LIN {X 0,Y 298.495,Z 251.301,A -85,B 0,C 180,E1 -16396.412,E2 -16396.412} C_VEL
LIN {X 0,Y 298.486,Z 251.3,A -85,B 0,C 180,E1 -16399.636,E2 -16399.636} C_VEL
LIN {X 0,Y 298.389,Z 251.313,A -85,B 0,C 180,E1 -16403.604,E2 -16403.604} C_VEL
LIN {X 0,Y 298.41,Z 251.315,A -85,B 0,C 180,E1 -16406.582,E2 -16406.582} C_VEL
LIN {X 0,Y 298.369,Z 251.315,A -85,B 0,C 180,E1 -16409.647,E2 -16409.647} C_VEL
LIN {X 0,Y 298.401,Z 251.314,A -85,B 0,C 180,E1 -16412.8,E2 -16412.8} C_VEL
LIN {X 0,Y 298.454,Z 251.307,A -85,B 0,C 180,E1 -16416.807,E2 -16416.807} C_VEL
LIN {X 0,Y 298.395,Z 251.314,A -85,B 0,C 180,E1 -16421.087,E2 -16421.087} C_VEL
LIN {X 0,Y 298.407,Z 251.311,A -85,B 0,C 180,E1 -16423.102,E2 -16423.102} C_VEL
LIN {X 0,Y 298.377,Z 251.316,A -85,B 0,C 180,E1 -16426.914,E2 -16426.914} C_VEL
LIN {X 0,Y 298.358,Z 251.318,A -85,B 0,C 180,E1 -16431.018,E2 -16431.018} C_VEL
LIN {X 0,Y 298.41,Z 251.316,A -85,B 0,C 180,E1 -16433.927,E2 -16433.927} C_VEL
LIN {X 0,Y 298.349,Z 251.319,A -85,B 0,C 180,E1 -16437.192,E2 -16437.192} C_VEL
LIN {X 0,Y 298.079,Z 251.351,A -85,B 0,C 180,E1 -16440.736,E2 -16440.736} C_VEL
LIN {X 0,Y 297.924,Z 251.374,A -85,B 0,C 180,E1 -16441.847,E2 -16441.847} C_VEL
LIN {X 0,Y 297.795,Z 253.558,A -85,B 0,C 180,E1 -16444.86,E2 -16444.86} C_VEL
LIN {X 0,Y 297.677,Z 255.967,A -85,B 0,C 180,E1 -16447.804,E2 -16447.804} C_VEL
LIN {X 0,Y 297.6,Z 258.252,A -85,B 0,C 180,E1 -16450.465,E2 -16450.465} C_VEL
LIN {X 0,Y 301.663,Z 271.623,A -85,B 0,C 180,E1 -16451.421,E2 -16451.421} C_VEL
LIN {X 0,Y 304.774,Z 284.38,A -85,B 0,C 180,E1 -16452.554,E2 -16452.554} C_VEL
LIN {X 0,Y 306.16,Z 292.534,A -85,B 0,C 180,E1 -16453.404,E2 -16453.404} C_VEL
LIN {X 0,Y 304.897,Z 304.106,A -85,B 0,C 180,E1 -16454.626,E2 -16454.626} C_VEL
LIN {X 0,Y 303.62,Z 314.955,A -85,B 0,C 180,E1 -16456.102,E2 -16456.102} C_VEL
LIN {X 0,Y 302.035,Z 325.56,A -85,B 0,C 180,E1 -16457.91,E2 -16457.91} C_VEL
LIN {X 0,Y 300.876,Z 333.375,A -85,B 0,C 180,E1 -16459.568,E2 -16459.568} C_VEL
LIN {X 0,Y 299.75,Z 341.018,A -85,B 0,C 180,E1 -16461.572,E2 -16461.572} C_VEL
LIN {X 0,Y 298.938,Z 346.239,A -85,B 0,C 180,E1 -16463.247,E2 -16463.247} C_VEL
LIN {X 0,Y 297.998,Z 351.328,A -85,B 0,C 180,E1 -16465.263,E2 -16465.263} C_VEL
LIN {X 0,Y 297.426,Z 355.273,A -85,B 0,C 180,E1 -16467.289,E2 -16467.289} C_VEL
LIN {X 0,Y 297.194,Z 357.306,A -85,B 0,C 180,E1 -16468.643,E2 -16468.643} C_VEL
LIN {X 0,Y 297.056,Z 358.924,A -85,B 0,C 180,E1 -16469.998,E2 -16469.998} C_VEL
LIN {X 0,Y 296.954,Z 360.15,A -85,B 0,C 180,E1 -16471.354,E2 -16471.354} C_VEL
LIN {X 0,Y 296.857,Z 360.979,A -85,B 0,C 180,E1 -16472.712,E2 -16472.712} C_VEL
LIN {X 0,Y 296.97,Z 361.408,A -85,B 0,C 180,E1 -16475.43,E2 -16475.43} C_VEL
LIN {X 0,Y 297.058,Z 361.061,A -85,B 0,C 180,E1 -16476.792,E2 -16476.792} C_VEL
LIN {X 0,Y 297.19,Z 360.323,A -85,B 0,C 180,E1 -16478.155,E2 -16478.155} C_VEL
LIN {X 0,Y 297.693,Z 357.573,A -85,B 0,C 180,E1 -16480.884,E2 -16480.884} C_VEL
LIN {X 0,Y 298.353,Z 354.392,A -85,B 0,C 180,E1 -16482.929,E2 -16482.929} C_VEL
LIN {X 0,Y 299.246,Z 350.14,A -85,B 0,C 180,E1 -16484.97,E2 -16484.97} C_VEL
LIN {X 0,Y 300.406,Z 344.691,A -85,B 0,C 180,E1 -16487.002,E2 -16487.002} C_VEL
LIN {X 0,Y 301.868,Z 337.861,A -85,B 0,C 180,E1 -16489.021,E2 -16489.021} C_VEL
LIN {X 0,Y 303.56,Z 329.278,A -85,B 0,C 180,E1 -16491.028,E2 -16491.028} C_VEL
LIN {X 0,Y 305.117,Z 320.347,A -85,B 0,C 180,E1 -16492.71,E2 -16492.71} C_VEL
LIN {X 0,Y 306.776,Z 310.709,A -85,B 0,C 180,E1 -16494.171,E2 -16494.171} C_VEL
LIN {X 0,Y 308.399,Z 299.995,A -85,B 0,C 180,E1 -16495.474,E2 -16495.474} C_VEL
LIN {X 0,Y 308.698,Z 295.769,A -85,B 0,C 180,E1 -16495.93,E2 -16495.93} C_VEL
LIN {X 0,Y 306.296,Z 284.543,A -85,B 0,C 180,E1 -16497.236,E2 -16497.236} C_VEL
LIN {X 0,Y 302.82,Z 272.388,A -85,B 0,C 180,E1 -16498.45,E2 -16498.45} C_VEL
LIN {X 0,Y 298.604,Z 261.16,A -85,B 0,C 180,E1 -16499.443,E2 -16499.443} C_VEL
LIN {X 0,Y 297.888,Z 258.687,A -85,B 0,C 180,E1 -16499.656,E2 -16499.656} C_VEL
LIN {X 0,Y 298.06,Z 256.149,A -85,B 0,C 180,E1 -16502.839,E2 -16502.839} C_VEL
LIN {X 0,Y 298.264,Z 253.165,A -85,B 0,C 180,E1 -16506.76,E2 -16506.76} C_VEL
LIN {X 0,Y 298.264,Z 251.331,A -85,B 0,C 180,E1 -16509.506,E2 -16509.506} C_VEL
LIN {X 0,Y 298.363,Z 251.321,A -85,B 0,C 180,E1 -16513.095,E2 -16513.095} C_VEL
LIN {X 0,Y 298.396,Z 251.317,A -85,B 0,C 180,E1 -16516.919,E2 -16516.919} C_VEL
LIN {X 0,Y 298.407,Z 251.314,A -85,B 0,C 180,E1 -16521.002,E2 -16521.002} C_VEL
LIN {X 0,Y 298.424,Z 251.31,A -85,B 0,C 180,E1 -16523.931,E2 -16523.931} C_VEL
LIN {X 0,Y 298.384,Z 251.317,A -85,B 0,C 180,E1 -16527.982,E2 -16527.982} C_VEL
LIN {X 0,Y 298.449,Z 251.307,A -85,B 0,C 180,E1 -16531.903,E2 -16531.903} C_VEL
LIN {X 0,Y 298.476,Z 251.305,A -85,B 0,C 180,E1 -16534.923,E2 -16534.923} C_VEL
LIN {X 0,Y 298.44,Z 251.31,A -85,B 0,C 180,E1 -16539.314,E2 -16539.314} C_VEL
LIN {X 0,Y 298.527,Z 251.299,A -85,B 0,C 180,E1 -16542.178,E2 -16542.178} C_VEL
LIN {X 0,Y 298.539,Z 251.294,A -85,B 0,C 180,E1 -16545.707,E2 -16545.707} C_VEL
LIN {X 0,Y 298.582,Z 251.294,A -85,B 0,C 180,E1 -16549.146,E2 -16549.146} C_VEL
LIN {X 0,Y 298.744,Z 251.272,A -85,B 0,C 180,E1 -16551.565,E2 -16551.565} C_VEL
LIN {X 0,Y 298.09,Z 251.356,A -85,B 0,C 180,E1 -16552.688,E2 -16552.688} C_VEL
LIN {X 0,Y 295.26,Z 251.712,A -85,B 0,C 180,E1 -16554.517,E2 -16554.517} C_VEL
LIN {X 0,Y 292.869,Z 252.008,A -85,B 0,C 180,E1 -16556.002,E2 -16556.002} C_VEL
LIN {X 0,Y 291.865,Z 252.131,A -85,B 0,C 180,E1 -16557.151,E2 -16557.151} C_VEL
LIN {X 0,Y 291.795,Z 252.137,A -85,B 0,C 180,E1 -16557.54,E2 -16557.54} C_VEL
LIN {X 0,Y 291.941,Z 252.12,A -85,B 0,C 180,E1 -16560,E2 -16560} C_VEL
LIN {X 0,Y 291.781,Z 252.14,A -85,B 0,C 180,E1 -16562.761,E2 -16562.761} C_VEL
LIN {X 0,Y 291.738,Z 252.145,A -85,B 0,C 180,E1 -16566.918,E2 -16566.918} C_VEL
LIN {X 0,Y 291.618,Z 252.16,A -85,B 0,C 180,E1 -16569.712,E2 -16569.712} C_VEL
LIN {X 0,Y 291.511,Z 252.173,A -85,B 0,C 180,E1 -16573.951,E2 -16573.951} C_VEL
LIN {X 0,Y 291.476,Z 252.176,A -85,B 0,C 180,E1 -16576.818,E2 -16576.818} C_VEL
LIN {X 0,Y 291.44,Z 252.179,A -85,B 0,C 180,E1 -16579.876,E2 -16579.876} C_VEL
LIN {X 0,Y 291.39,Z 252.188,A -85,B 0,C 180,E1 -16584.206,E2 -16584.206} C_VEL
LIN {X 0,Y 291.415,Z 252.185,A -85,B 0,C 180,E1 -16587.272,E2 -16587.272} C_VEL
LIN {X 0,Y 291.331,Z 252.197,A -85,B 0,C 180,E1 -16590.437,E2 -16590.437} C_VEL
LIN {X 0,Y 291.336,Z 252.196,A -85,B 0,C 180,E1 -16593.699,E2 -16593.699} C_VEL
LIN {X 0,Y 291.416,Z 252.319,A -85,B 0,C 180,E1 -16596.863,E2 -16596.863} C_VEL
LIN {X 0,Y 292.017,Z 256.126,A -85,B 0,C 180,E1 -16600.527,E2 -16600.527} C_VEL
LIN {X 0,Y 292.801,Z 260.152,A -85,B 0,C 180,E1 -16604.113,E2 -16604.113} C_VEL
LIN {X 0,Y 293.64,Z 264.805,A -85,B 0,C 180,E1 -16607.924,E2 -16607.924} C_VEL
LIN {X 0,Y 294.327,Z 268.492,A -85,B 0,C 180,E1 -16610.771,E2 -16610.771} C_VEL
LIN {X 0,Y 294.514,Z 272.114,A -85,B 0,C 180,E1 -16613.378,E2 -16613.378} C_VEL
LIN {X 0,Y 293.527,Z 277.438,A -85,B 0,C 180,E1 -16616.931,E2 -16616.931} C_VEL
LIN {X 0,Y 292.414,Z 284.163,A -85,B 0,C 180,E1 -16621.272,E2 -16621.272} C_VEL
LIN {X 0,Y 291.705,Z 288.494,A -85,B 0,C 180,E1 -16624.014,E2 -16624.014} C_VEL
LIN {X 0,Y 295.156,Z 303.237,A -85,B 0,C 180,E1 -16625.062,E2 -16625.062} C_VEL
LIN {X 0,Y 297.245,Z 315.455,A -85,B 0,C 180,E1 -16626.118,E2 -16626.118} C_VEL
LIN {X 0,Y 298.415,Z 327.56,A -85,B 0,C 180,E1 -16627.354,E2 -16627.354} C_VEL
LIN {X 0,Y 298.729,Z 339.369,A -85,B 0,C 180,E1 -16628.797,E2 -16628.797} C_VEL
LIN {X 0,Y 296.902,Z 350.121,A -85,B 0,C 180,E1 -16630.289,E2 -16630.289} C_VEL
LIN {X 0,Y 295.152,Z 359.818,A -85,B 0,C 180,E1 -16631.97,E2 -16631.97} C_VEL
LIN {X 0,Y 293.752,Z 367.79,A -85,B 0,C 180,E1 -16633.675,E2 -16633.675} C_VEL
LIN {X 0,Y 292.298,Z 375.615,A -85,B 0,C 180,E1 -16635.735,E2 -16635.735} C_VEL
LIN {X 0,Y 290.944,Z 382.812,A -85,B 0,C 180,E1 -16638.154,E2 -16638.154} C_VEL
LIN {X 0,Y 290.222,Z 387.639,A -85,B 0,C 180,E1 -16640.243,E2 -16640.243} C_VEL
LIN {X 0,Y 289.804,Z 391.357,A -85,B 0,C 180,E1 -16642.337,E2 -16642.337} C_VEL
LIN {X 0,Y 289.624,Z 394.066,A -85,B 0,C 180,E1 -16644.432,E2 -16644.432} C_VEL
LIN {X 0,Y 289.579,Z 395.353,A -85,B 0,C 180,E1 -16645.827,E2 -16645.827} C_VEL
LIN {X 0,Y 289.548,Z 396.233,A -85,B 0,C 180,E1 -16647.22,E2 -16647.22} C_VEL
LIN {X 0,Y 289.693,Z 396.729,A -85,B 0,C 180,E1 -16650.002,E2 -16650.002} C_VEL
LIN {X 0,Y 289.608,Z 396.378,A -85,B 0,C 180,E1 -16651.393,E2 -16651.393} C_VEL
LIN {X 0,Y 289.568,Z 395.633,A -85,B 0,C 180,E1 -16652.784,E2 -16652.784} C_VEL
LIN {X 0,Y 289.605,Z 394.441,A -85,B 0,C 180,E1 -16654.177,E2 -16654.177} C_VEL
LIN {X 0,Y 289.638,Z 392.512,A -85,B 0,C 180,E1 -16655.813,E2 -16655.813} C_VEL
LIN {X 0,Y 289.919,Z 388.286,A -85,B 0,C 180,E1 -16658.365,E2 -16658.365} C_VEL
LIN {X 0,Y 290.444,Z 383.58,A -85,B 0,C 180,E1 -16660.458,E2 -16660.458} C_VEL
LIN {X 0,Y 291.385,Z 376.481,A -85,B 0,C 180,E1 -16662.893,E2 -16662.893} C_VEL
LIN {X 0,Y 292.543,Z 368.803,A -85,B 0,C 180,E1 -16664.969,E2 -16664.969} C_VEL
LIN {X 0,Y 293.742,Z 360.95,A -85,B 0,C 180,E1 -16666.687,E2 -16666.687} C_VEL
LIN {X 0,Y 295.134,Z 351.353,A -85,B 0,C 180,E1 -16668.394,E2 -16668.394} C_VEL
LIN {X 0,Y 296.77,Z 340.732,A -85,B 0,C 180,E1 -16669.905,E2 -16669.905} C_VEL
LIN {X 0,Y 297.183,Z 336.584,A -85,B 0,C 180,E1 -16670.417,E2 -16670.417} C_VEL
LIN {X 0,Y 296.404,Z 324.766,A -85,B 0,C 180,E1 -16671.772,E2 -16671.772} C_VEL
LIN {X 0,Y 295.302,Z 312.997,A -85,B 0,C 180,E1 -16672.858,E2 -16672.858} C_VEL
LIN {X 0,Y 293.429,Z 300.224,A -85,B 0,C 180,E1 -16673.794,E2 -16673.794} C_VEL
LIN {X 0,Y 291.24,Z 288.858,A -85,B 0,C 180,E1 -16674.459,E2 -16674.459} C_VEL
LIN {X 0,Y 292.173,Z 281.913,A -85,B 0,C 180,E1 -16678.758,E2 -16678.758} C_VEL
LIN {X 0,Y 293.275,Z 275.145,A -85,B 0,C 180,E1 -16682.993,E2 -16682.993} C_VEL
LIN {X 0,Y 293.926,Z 271.096,A -85,B 0,C 180,E1 -16685.613,E2 -16685.613} C_VEL
LIN {X 0,Y 294.053,Z 267.61,A -85,B 0,C 180,E1 -16687.934,E2 -16687.934} C_VEL
LIN {X 0,Y 293.376,Z 263.132,A -85,B 0,C 180,E1 -16691.125,E2 -16691.125} C_VEL
LIN {X 0,Y 292.462,Z 258.16,A -85,B 0,C 180,E1 -16694.976,E2 -16694.976} C_VEL
LIN {X 0,Y 291.512,Z 252.834,A -85,B 0,C 180,E1 -16699.388,E2 -16699.388} C_VEL
LIN {X 0,Y 291.377,Z 252.193,A -85,B 0,C 180,E1 -16700.006,E2 -16700.006} C_VEL
LIN {X 0,Y 291.411,Z 252.187,A -85,B 0,C 180,E1 -16702.92,E2 -16702.92} C_VEL
LIN {X 0,Y 291.351,Z 252.194,A -85,B 0,C 180,E1 -16706.302,E2 -16706.302} C_VEL
LIN {X 0,Y 291.377,Z 252.191,A -85,B 0,C 180,E1 -16710.267,E2 -16710.267} C_VEL
LIN {X 0,Y 291.385,Z 252.19,A -85,B 0,C 180,E1 -16714.269,E2 -16714.269} C_VEL
LIN {X 0,Y 291.379,Z 252.187,A -85,B 0,C 180,E1 -16717.299,E2 -16717.299} C_VEL
LIN {X 0,Y 291.414,Z 252.187,A -85,B 0,C 180,E1 -16720.267,E2 -16720.267} C_VEL
LIN {X 0,Y 291.482,Z 252.176,A -85,B 0,C 180,E1 -16724.683,E2 -16724.683} C_VEL
LIN {X 0,Y 291.534,Z 252.169,A -85,B 0,C 180,E1 -16728.881,E2 -16728.881} C_VEL
LIN {X 0,Y 291.676,Z 252.155,A -85,B 0,C 180,E1 -16731.688,E2 -16731.688} C_VEL
LIN {X 0,Y 291.63,Z 252.157,A -85,B 0,C 180,E1 -16734.468,E2 -16734.468} C_VEL
LIN {X 0,Y 291.895,Z 252.123,A -85,B 0,C 180,E1 -16738.621,E2 -16738.621} C_VEL
LIN {X 0,Y 291.889,Z 252.126,A -85,B 0,C 180,E1 -16741.38,E2 -16741.38} C_VEL
LIN {X 0,Y 291.693,Z 252.15,A -85,B 0,C 180,E1 -16746.919,E2 -16746.919} C_VEL
LIN {X 0,Y 291.577,Z 252.162,A -85,B 0,C 180,E1 -16749.714,E2 -16749.714} C_VEL
LIN {X 0,Y 291.524,Z 252.168,A -85,B 0,C 180,E1 -16753.95,E2 -16753.95} C_VEL
LIN {X 0,Y 291.442,Z 252.182,A -85,B 0,C 180,E1 -16756.821,E2 -16756.821} C_VEL
LIN {X 0,Y 291.433,Z 252.178,A -85,B 0,C 180,E1 -16759.86,E2 -16759.86} C_VEL
LIN {X 0,Y 291.334,Z 252.193,A -85,B 0,C 180,E1 -16764.211,E2 -16764.211} C_VEL
LIN {X 0,Y 291.34,Z 252.193,A -85,B 0,C 180,E1 -16767.28,E2 -16767.28} C_VEL
LIN {X 0,Y 291.312,Z 252.198,A -85,B 0,C 180,E1 -16770.44,E2 -16770.44} C_VEL
LIN {X 0,Y 291.352,Z 252.19,A -85,B 0,C 180,E1 -16773.698,E2 -16773.698} C_VEL
LIN {X 0,Y 291.384,Z 252.186,A -85,B 0,C 180,E1 -16777.253,E2 -16777.253} C_VEL
LIN {X 0,Y 291.34,Z 252.195,A -85,B 0,C 180,E1 -16780.642,E2 -16780.642} C_VEL
LIN {X 0,Y 291.298,Z 252.2,A -85,B 0,C 180,E1 -16784.401,E2 -16784.401} C_VEL
LIN {X 0,Y 291.301,Z 252.2,A -85,B 0,C 180,E1 -16788.411,E2 -16788.411} C_VEL
LIN {X 0,Y 291.392,Z 252.186,A -85,B 0,C 180,E1 -16792.915,E2 -16792.915} C_VEL
LIN {X 0,Y 291.328,Z 252.194,A -85,B 0,C 180,E1 -16796.297,E2 -16796.297} C_VEL
LIN {X 0,Y 291.106,Z 252.221,A -85,B 0,C 180,E1 -16799.534,E2 -16799.534} C_VEL
LIN {X 0,Y 290.966,Z 252.238,A -85,B 0,C 180,E1 -16801.111,E2 -16801.111} C_VEL
LIN {X 0,Y 290.841,Z 252.791,A -85,B 0,C 180,E1 -16802.667,E2 -16802.667} C_VEL
LIN {X 0,Y 290.667,Z 256.033,A -85,B 0,C 180,E1 -16806.752,E2 -16806.752} C_VEL
LIN {X 0,Y 290.568,Z 258.744,A -85,B 0,C 180,E1 -16809.906,E2 -16809.906} C_VEL
LIN {X 0,Y 294.61,Z 271.745,A -85,B 0,C 180,E1 -16810.872,E2 -16810.872} C_VEL
LIN {X 0,Y 297.663,Z 283.982,A -85,B 0,C 180,E1 -16811.988,E2 -16811.988} C_VEL
LIN {X 0,Y 299.429,Z 293.541,A -85,B 0,C 180,E1 -16813.017,E2 -16813.017} C_VEL
LIN {X 0,Y 298.114,Z 305.01,A -85,B 0,C 180,E1 -16814.268,E2 -16814.268} C_VEL
LIN {X 0,Y 296.773,Z 315.748,A -85,B 0,C 180,E1 -16815.775,E2 -16815.775} C_VEL
LIN {X 0,Y 295.139,Z 326.292,A -85,B 0,C 180,E1 -16817.623,E2 -16817.623} C_VEL
LIN {X 0,Y 293.944,Z 334.054,A -85,B 0,C 180,E1 -16819.32,E2 -16819.32} C_VEL
LIN {X 0,Y 292.75,Z 341.637,A -85,B 0,C 180,E1 -16821.369,E2 -16821.369} C_VEL
LIN {X 0,Y 291.525,Z 348.63,A -85,B 0,C 180,E1 -16823.77,E2 -16823.77} C_VEL
LIN {X 0,Y 290.747,Z 353.286,A -85,B 0,C 180,E1 -16825.839,E2 -16825.839} C_VEL
LIN {X 0,Y 290.225,Z 356.849,A -85,B 0,C 180,E1 -16827.916,E2 -16827.916} C_VEL
LIN {X 0,Y 289.981,Z 359.412,A -85,B 0,C 180,E1 -16829.998,E2 -16829.998} C_VEL
LIN {X 0,Y 289.861,Z 360.626,A -85,B 0,C 180,E1 -16831.387,E2 -16831.387} C_VEL
LIN {X 0,Y 289.772,Z 361.427,A -85,B 0,C 180,E1 -16832.778,E2 -16832.778} C_VEL
LIN {X 0,Y 289.906,Z 361.828,A -85,B 0,C 180,E1 -16835.563,E2 -16835.563} C_VEL
LIN {X 0,Y 289.996,Z 361.469,A -85,B 0,C 180,E1 -16836.958,E2 -16836.958} C_VEL
LIN {X 0,Y 290.128,Z 360.706,A -85,B 0,C 180,E1 -16838.355,E2 -16838.355} C_VEL
LIN {X 0,Y 290.68,Z 357.926,A -85,B 0,C 180,E1 -16841.15,E2 -16841.15} C_VEL
LIN {X 0,Y 291.399,Z 354.714,A -85,B 0,C 180,E1 -16843.243,E2 -16843.243} C_VEL
LIN {X 0,Y 292.34,Z 350.43,A -85,B 0,C 180,E1 -16845.332,E2 -16845.332} C_VEL
LIN {X 0,Y 293.568,Z 344.946,A -85,B 0,C 180,E1 -16847.41,E2 -16847.41} C_VEL
LIN {X 0,Y 295.116,Z 338.074,A -85,B 0,C 180,E1 -16849.473,E2 -16849.473} C_VEL
LIN {X 0,Y 296.91,Z 329.424,A -85,B 0,C 180,E1 -16851.522,E2 -16851.522} C_VEL
LIN {X 0,Y 298.437,Z 321.024,A -85,B 0,C 180,E1 -16853.137,E2 -16853.137} C_VEL
LIN {X 0,Y 300.28,Z 310.729,A -85,B 0,C 180,E1 -16854.729,E2 -16854.729} C_VEL
LIN {X 0,Y 301.951,Z 299.88,A -85,B 0,C 180,E1 -16856.058,E2 -16856.058} C_VEL
LIN {X 0,Y 302.019,Z 296.95,A -85,B 0,C 180,E1 -16856.394,E2 -16856.394} C_VEL
LIN {X 0,Y 299.713,Z 286.068,A -85,B 0,C 180,E1 -16857.723,E2 -16857.723} C_VEL
LIN {X 0,Y 296.345,Z 274.182,A -85,B 0,C 180,E1 -16858.977,E2 -16858.977} C_VEL
LIN {X 0,Y 291.861,Z 262.102,A -85,B 0,C 180,E1 -16860.099,E2 -16860.099} C_VEL
LIN {X 0,Y 290.879,Z 259.15,A -85,B 0,C 180,E1 -16860.354,E2 -16860.354} C_VEL
LIN {X 0,Y 291.079,Z 256.531,A -85,B 0,C 180,E1 -16863.731,E2 -16863.731} C_VEL
LIN {X 0,Y 291.249,Z 253.962,A -85,B 0,C 180,E1 -16867.22,E2 -16867.22} C_VEL
LIN {X 0,Y 291.257,Z 252.385,A -85,B 0,C 180,E1 -16869.452,E2 -16869.452} C_VEL
LIN {X 0,Y 291.277,Z 252.203,A -85,B 0,C 180,E1 -16872.497,E2 -16872.497} C_VEL
LIN {X 0,Y 291.302,Z 252.201,A -85,B 0,C 180,E1 -16876.364,E2 -16876.364} C_VEL
LIN {X 0,Y 291.379,Z 252.191,A -85,B 0,C 180,E1 -16880.515,E2 -16880.515} C_VEL
LIN {X 0,Y 291.417,Z 252.183,A -85,B 0,C 180,E1 -16882.921,E2 -16882.921} C_VEL
LIN {X 0,Y 291.336,Z 252.192,A -85,B 0,C 180,E1 -16886.3,E2 -16886.3} C_VEL
LIN {X 0,Y 291.374,Z 252.189,A -85,B 0,C 180,E1 -16890.26,E2 -16890.26} C_VEL
LIN {X 0,Y 291.405,Z 252.189,A -85,B 0,C 180,E1 -16894.271,E2 -16894.271} C_VEL
LIN {X 0,Y 291.372,Z 252.191,A -85,B 0,C 180,E1 -16897.298,E2 -16897.298} C_VEL
LIN {X 0,Y 291.448,Z 252.181,A -85,B 0,C 180,E1 -16900.269,E2 -16900.269} C_VEL
LIN {X 0,Y 291.545,Z 252.169,A -85,B 0,C 180,E1 -16904.623,E2 -16904.623} C_VEL
LIN {X 0,Y 291.526,Z 252.171,A -85,B 0,C 180,E1 -16908.88,E2 -16908.88} C_VEL
LIN {X 0,Y 291.7,Z 252.15,A -85,B 0,C 180,E1 -16911.688,E2 -16911.688} C_VEL
LIN {X 0,Y 291.625,Z 252.16,A -85,B 0,C 180,E1 -16914.468,E2 -16914.468} C_VEL
LIN {X 0,Y 291.795,Z 252.137,A -85,B 0,C 180,E1 -16917.54,E2 -16917.54} C_VEL
LIN {X 0,Y 291.168,Z 252.217,A -85,B 0,C 180,E1 -16918.694,E2 -16918.694} C_VEL
LIN {X 0,Y 288.341,Z 252.569,A -85,B 0,C 180,E1 -16920.573,E2 -16920.573} C_VEL
LIN {X 0,Y 284.987,Z 252.986,A -85,B 0,C 180,E1 -16922.88,E2 -16922.88} C_VEL
LIN {X 0,Y 284.575,Z 253.034,A -85,B 0,C 180,E1 -16923.679,E2 -16923.679} C_VEL
LIN {X 0,Y 284.69,Z 253.023,A -85,B 0,C 180,E1 -16927.09,E2 -16927.09} C_VEL
LIN {X 0,Y 284.555,Z 253.04,A -85,B 0,C 180,E1 -16929.956,E2 -16929.956} C_VEL
LIN {X 0,Y 284.47,Z 253.048,A -85,B 0,C 180,E1 -16934.303,E2 -16934.303} C_VEL
LIN {X 0,Y 284.415,Z 253.058,A -85,B 0,C 180,E1 -16937.249,E2 -16937.249} C_VEL
LIN {X 0,Y 284.368,Z 253.063,A -85,B 0,C 180,E1 -16940.243,E2 -16940.243} C_VEL
LIN {X 0,Y 284.359,Z 253.065,A -85,B 0,C 180,E1 -16943.876,E2 -16943.876} C_VEL
LIN {X 0,Y 284.388,Z 253.06,A -85,B 0,C 180,E1 -16947.175,E2 -16947.175} C_VEL
LIN {X 0,Y 284.289,Z 253.073,A -85,B 0,C 180,E1 -16951.275,E2 -16951.275} C_VEL
LIN {X 0,Y 284.332,Z 253.064,A -85,B 0,C 180,E1 -16955.349,E2 -16955.349} C_VEL
LIN {X 0,Y 284.35,Z 253.206,A -85,B 0,C 180,E1 -16956.09,E2 -16956.09} C_VEL
LIN {X 0,Y 285.031,Z 257.246,A -85,B 0,C 180,E1 -16960.153,E2 -16960.153} C_VEL
LIN {X 0,Y 285.946,Z 262.067,A -85,B 0,C 180,E1 -16964.543,E2 -16964.543} C_VEL
LIN {X 0,Y 286.818,Z 266.953,A -85,B 0,C 180,E1 -16968.582,E2 -16968.582} C_VEL
LIN {X 0,Y 287.436,Z 270.659,A -85,B 0,C 180,E1 -16971.483,E2 -16971.483} C_VEL
LIN {X 0,Y 287.374,Z 273.855,A -85,B 0,C 180,E1 -16973.808,E2 -16973.808} C_VEL
LIN {X 0,Y 286.624,Z 277.769,A -85,B 0,C 180,E1 -16976.479,E2 -16976.479} C_VEL
LIN {X 0,Y 285.488,Z 283.813,A -85,B 0,C 180,E1 -16980.508,E2 -16980.508} C_VEL
LIN {X 0,Y 284.815,Z 288.181,A -85,B 0,C 180,E1 -16983.309,E2 -16983.309} C_VEL
LIN {X 0,Y 287.416,Z 298.87,A -85,B 0,C 180,E1 -16984.06,E2 -16984.06} C_VEL
LIN {X 0,Y 289.847,Z 311.024,A -85,B 0,C 180,E1 -16985.093,E2 -16985.093} C_VEL
LIN {X 0,Y 291.332,Z 322.541,A -85,B 0,C 180,E1 -16986.24,E2 -16986.24} C_VEL
LIN {X 0,Y 291.907,Z 333.646,A -85,B 0,C 180,E1 -16987.532,E2 -16987.532} C_VEL
LIN {X 0,Y 291.912,Z 340.559,A -85,B 0,C 180,E1 -16988.462,E2 -16988.462} C_VEL
LIN {X 0,Y 290.006,Z 351.033,A -85,B 0,C 180,E1 -16989.985,E2 -16989.985} C_VEL
LIN {X 0,Y 288.165,Z 360.713,A -85,B 0,C 180,E1 -16991.751,E2 -16991.751} C_VEL
LIN {X 0,Y 286.626,Z 368.947,A -85,B 0,C 180,E1 -16993.624,E2 -16993.624} C_VEL
LIN {X 0,Y 285.155,Z 376.45,A -85,B 0,C 180,E1 -16995.734,E2 -16995.734} C_VEL
LIN {X 0,Y 283.944,Z 382.493,A -85,B 0,C 180,E1 -16997.857,E2 -16997.857} C_VEL
LIN {X 0,Y 283.195,Z 387.297,A -85,B 0,C 180,E1 -16999.998,E2 -16999.998} C_VEL
LIN {X 0,Y 282.737,Z 390.993,A -85,B 0,C 180,E1 -17002.144,E2 -17002.144} C_VEL
LIN {X 0,Y 282.541,Z 393.682,A -85,B 0,C 180,E1 -17004.292,E2 -17004.292} C_VEL
LIN {X 0,Y 282.5,Z 394.959,A -85,B 0,C 180,E1 -17005.722,E2 -17005.722} C_VEL
LIN {X 0,Y 282.475,Z 395.824,A -85,B 0,C 180,E1 -17007.15,E2 -17007.15} C_VEL
LIN {X 0,Y 282.604,Z 396.297,A -85,B 0,C 180,E1 -17010.002,E2 -17010.002} C_VEL
LIN {X 0,Y 282.521,Z 395.936,A -85,B 0,C 180,E1 -17011.428,E2 -17011.428} C_VEL
LIN {X 0,Y 282.494,Z 395.177,A -85,B 0,C 180,E1 -17012.854,E2 -17012.854} C_VEL
LIN {X 0,Y 282.522,Z 393.968,A -85,B 0,C 180,E1 -17014.282,E2 -17014.282} C_VEL
LIN {X 0,Y 282.559,Z 392.251,A -85,B 0,C 180,E1 -17015.784,E2 -17015.784} C_VEL
LIN {X 0,Y 282.747,Z 389.076,A -85,B 0,C 180,E1 -17017.859,E2 -17017.859} C_VEL
LIN {X 0,Y 283.217,Z 384.731,A -85,B 0,C 180,E1 -17020.005,E2 -17020.005} C_VEL
LIN {X 0,Y 284.069,Z 378.16,A -85,B 0,C 180,E1 -17022.504,E2 -17022.504} C_VEL
LIN {X 0,Y 285.26,Z 370.955,A -85,B 0,C 180,E1 -17024.629,E2 -17024.629} C_VEL
LIN {X 0,Y 286.66,Z 361.977,A -85,B 0,C 180,E1 -17026.745,E2 -17026.745} C_VEL
LIN {X 0,Y 288.056,Z 352.767,A -85,B 0,C 180,E1 -17028.494,E2 -17028.494} C_VEL
LIN {X 0,Y 289.65,Z 342.578,A -85,B 0,C 180,E1 -17030.045,E2 -17030.045} C_VEL
LIN {X 0,Y 290.295,Z 337.231,A -85,B 0,C 180,E1 -17030.738,E2 -17030.738} C_VEL
LIN {X 0,Y 289.54,Z 325.291,A -85,B 0,C 180,E1 -17032.166,E2 -17032.166} C_VEL
LIN {X 0,Y 288.485,Z 313.149,A -85,B 0,C 180,E1 -17033.334,E2 -17033.334} C_VEL
LIN {X 0,Y 286.603,Z 300.298,A -85,B 0,C 180,E1 -17034.319,E2 -17034.319} C_VEL
LIN {X 0,Y 284.248,Z 288.415,A -85,B 0,C 180,E1 -17035.052,E2 -17035.052} C_VEL
LIN {X 0,Y 285.294,Z 281.424,A -85,B 0,C 180,E1 -17039.519,E2 -17039.519} C_VEL
LIN {X 0,Y 286.334,Z 275.364,A -85,B 0,C 180,E1 -17043.434,E2 -17043.434} C_VEL
LIN {X 0,Y 287.068,Z 270.268,A -85,B 0,C 180,E1 -17046.858,E2 -17046.858} C_VEL
LIN {X 0,Y 287.02,Z 268.038,A -85,B 0,C 180,E1 -17048.413,E2 -17048.413} C_VEL
LIN {X 0,Y 286.291,Z 263.878,A -85,B 0,C 180,E1 -17051.517,E2 -17051.517} C_VEL
LIN {X 0,Y 285.323,Z 258.682,A -85,B 0,C 180,E1 -17055.59,E2 -17055.59} C_VEL
LIN {X 0,Y 284.426,Z 253.592,A -85,B 0,C 180,E1 -17060.026,E2 -17060.026} C_VEL
LIN {X 0,Y 284.329,Z 253.07,A -85,B 0,C 180,E1 -17060.699,E2 -17060.699} C_VEL
LIN {X 0,Y 284.348,Z 253.067,A -85,B 0,C 180,E1 -17064.653,E2 -17064.653} C_VEL
LIN {X 0,Y 284.294,Z 253.072,A -85,B 0,C 180,E1 -17068.725,E2 -17068.725} C_VEL
LIN {X 0,Y 284.299,Z 253.071,A -85,B 0,C 180,E1 -17071.986,E2 -17071.986} C_VEL
LIN {X 0,Y 284.334,Z 253.069,A -85,B 0,C 180,E1 -17076.145,E2 -17076.145} C_VEL
LIN {X 0,Y 284.384,Z 253.062,A -85,B 0,C 180,E1 -17079.905,E2 -17079.905} C_VEL
LIN {X 0,Y 284.44,Z 253.054,A -85,B 0,C 180,E1 -17084.504,E2 -17084.504} C_VEL
LIN {X 0,Y 284.466,Z 253.05,A -85,B 0,C 180,E1 -17088.601,E2 -17088.601} C_VEL
LIN {X 0,Y 284.63,Z 253.031,A -85,B 0,C 180,E1 -17091.48,E2 -17091.48} C_VEL
LIN {X 0,Y 284.6,Z 253.033,A -85,B 0,C 180,E1 -17094.331,E2 -17094.331} C_VEL
LIN {X 0,Y 284.862,Z 252.999,A -85,B 0,C 180,E1 -17098.586,E2 -17098.586} C_VEL
LIN {X 0,Y 284.855,Z 253.002,A -85,B 0,C 180,E1 -17101.414,E2 -17101.414} C_VEL
LIN {X 0,Y 284.648,Z 253.028,A -85,B 0,C 180,E1 -17107.091,E2 -17107.091} C_VEL
LIN {X 0,Y 284.523,Z 253.04,A -85,B 0,C 180,E1 -17109.957,E2 -17109.957} C_VEL
LIN {X 0,Y 284.472,Z 253.046,A -85,B 0,C 180,E1 -17114.304,E2 -17114.304} C_VEL
LIN {X 0,Y 284.371,Z 253.063,A -85,B 0,C 180,E1 -17118.741,E2 -17118.741} C_VEL
LIN {X 0,Y 284.311,Z 253.068,A -85,B 0,C 180,E1 -17121.765,E2 -17121.765} C_VEL
LIN {X 0,Y 284.291,Z 253.072,A -85,B 0,C 180,E1 -17124.851,E2 -17124.851} C_VEL
LIN {X 0,Y 284.272,Z 253.073,A -85,B 0,C 180,E1 -17128.017,E2 -17128.017} C_VEL
LIN {X 0,Y 284.287,Z 253.071,A -85,B 0,C 180,E1 -17131.276,E2 -17131.276} C_VEL
LIN {X 0,Y 284.349,Z 253.063,A -85,B 0,C 180,E1 -17135.347,E2 -17135.347} C_VEL
LIN {X 0,Y 284.32,Z 253.069,A -85,B 0,C 180,E1 -17138.168,E2 -17138.168} C_VEL
LIN {X 0,Y 284.277,Z 253.076,A -85,B 0,C 180,E1 -17142.123,E2 -17142.123} C_VEL
LIN {X 0,Y 284.245,Z 253.08,A -85,B 0,C 180,E1 -17146.185,E2 -17146.185} C_VEL
LIN {X 0,Y 284.262,Z 253.078,A -85,B 0,C 180,E1 -17150.035,E2 -17150.035} C_VEL
LIN {X 0,Y 284.322,Z 253.069,A -85,B 0,C 180,E1 -17153.61,E2 -17153.61} C_VEL
LIN {X 0,Y 284.243,Z 253.076,A -85,B 0,C 180,E1 -17157.211,E2 -17157.211} C_VEL
LIN {X 0,Y 284.016,Z 253.103,A -85,B 0,C 180,E1 -17160.335,E2 -17160.335} C_VEL
LIN {X 0,Y 283.827,Z 253.24,A -85,B 0,C 180,E1 -17161.933,E2 -17161.933} C_VEL
LIN {X 0,Y 283.689,Z 255.673,A -85,B 0,C 180,E1 -17165.091,E2 -17165.091} C_VEL
LIN {X 0,Y 283.539,Z 258.972,A -85,B 0,C 180,E1 -17169.181,E2 -17169.181} C_VEL
LIN {X 0,Y 283.556,Z 259.174,A -85,B 0,C 180,E1 -17169.316,E2 -17169.316} C_VEL
LIN {X 0,Y 287.672,Z 272.213,A -85,B 0,C 180,E1 -17170.326,E2 -17170.326} C_VEL
LIN {X 0,Y 290.573,Z 283.578,A -85,B 0,C 180,E1 -17171.395,E2 -17171.395} C_VEL
LIN {X 0,Y 292.681,Z 294.583,A -85,B 0,C 180,E1 -17172.614,E2 -17172.614} C_VEL
LIN {X 0,Y 291.343,Z 305.891,A -85,B 0,C 180,E1 -17173.892,E2 -17173.892} C_VEL
LIN {X 0,Y 289.955,Z 316.54,A -85,B 0,C 180,E1 -17175.433,E2 -17175.433} C_VEL
LIN {X 0,Y 288.258,Z 327.021,A -85,B 0,C 180,E1 -17177.323,E2 -17177.323} C_VEL
LIN {X 0,Y 287.019,Z 334.726,A -85,B 0,C 180,E1 -17179.059,E2 -17179.059} C_VEL
LIN {X 0,Y 285.754,Z 342.255,A -85,B 0,C 180,E1 -17181.156,E2 -17181.156} C_VEL
LIN {X 0,Y 284.902,Z 347.416,A -85,B 0,C 180,E1 -17182.913,E2 -17182.913} C_VEL
LIN {X 0,Y 283.931,Z 352.426,A -85,B 0,C 180,E1 -17185.028,E2 -17185.028} C_VEL
LIN {X 0,Y 283.332,Z 356.311,A -85,B 0,C 180,E1 -17187.154,E2 -17187.154} C_VEL
LIN {X 0,Y 283.085,Z 358.309,A -85,B 0,C 180,E1 -17188.575,E2 -17188.575} C_VEL
LIN {X 0,Y 282.907,Z 359.901,A -85,B 0,C 180,E1 -17189.998,E2 -17189.998} C_VEL
LIN {X 0,Y 282.769,Z 361.101,A -85,B 0,C 180,E1 -17191.422,E2 -17191.422} C_VEL
LIN {X 0,Y 282.757,Z 362.248,A -85,B 0,C 180,E1 -17194.274,E2 -17194.274} C_VEL
LIN {X 0,Y 282.888,Z 362.109,A -85,B 0,C 180,E1 -17196.406,E2 -17196.406} C_VEL
LIN {X 0,Y 283.085,Z 361.085,A -85,B 0,C 180,E1 -17198.564,E2 -17198.564} C_VEL
LIN {X 0,Y 283.689,Z 358.277,A -85,B 0,C 180,E1 -17201.429,E2 -17201.429} C_VEL
LIN {X 0,Y 284.458,Z 355.036,A -85,B 0,C 180,E1 -17203.572,E2 -17203.572} C_VEL
LIN {X 0,Y 285.45,Z 350.72,A -85,B 0,C 180,E1 -17205.711,E2 -17205.711} C_VEL
LIN {X 0,Y 286.779,Z 345.2,A -85,B 0,C 180,E1 -17207.836,E2 -17207.836} C_VEL
LIN {X 0,Y 288.404,Z 338.28,A -85,B 0,C 180,E1 -17209.945,E2 -17209.945} C_VEL
LIN {X 0,Y 290.285,Z 329.571,A -85,B 0,C 180,E1 -17212.038,E2 -17212.038} C_VEL
LIN {X 0,Y 292.069,Z 320.038,A -85,B 0,C 180,E1 -17213.88,E2 -17213.88} C_VEL
LIN {X 0,Y 294.034,Z 309.492,A -85,B 0,C 180,E1 -17215.48,E2 -17215.48} C_VEL
LIN {X 0,Y 295.531,Z 299.762,A -85,B 0,C 180,E1 -17216.668,E2 -17216.668} C_VEL
LIN {X 0,Y 293.744,Z 289.959,A -85,B 0,C 180,E1 -17217.935,E2 -17217.935} C_VEL
LIN {X 0,Y 290.847,Z 278.963,A -85,B 0,C 180,E1 -17219.199,E2 -17219.199} C_VEL
LIN {X 0,Y 286.926,Z 267.736,A -85,B 0,C 180,E1 -17220.355,E2 -17220.355} C_VEL
LIN {X 0,Y 283.969,Z 259.916,A -85,B 0,C 180,E1 -17221.058,E2 -17221.058} C_VEL
LIN {X 0,Y 283.907,Z 259.616,A -85,B 0,C 180,E1 -17221.083,E2 -17221.083} C_VEL
LIN {X 0,Y 284.102,Z 256.907,A -85,B 0,C 180,E1 -17224.675,E2 -17224.675} C_VEL
LIN {X 0,Y 284.233,Z 254.407,A -85,B 0,C 180,E1 -17228.179,E2 -17228.179} C_VEL
LIN {X 0,Y 284.215,Z 253.157,A -85,B 0,C 180,E1 -17230.007,E2 -17230.007} C_VEL
LIN {X 0,Y 284.226,Z 253.082,A -85,B 0,C 180,E1 -17234.186,E2 -17234.186} C_VEL
LIN {X 0,Y 284.265,Z 253.078,A -85,B 0,C 180,E1 -17238.123,E2 -17238.123} C_VEL
LIN {X 0,Y 284.327,Z 253.069,A -85,B 0,C 180,E1 -17242.273,E2 -17242.273} C_VEL
LIN {X 0,Y 284.315,Z 253.07,A -85,B 0,C 180,E1 -17245.351,E2 -17245.351} C_VEL
LIN {X 0,Y 284.285,Z 253.071,A -85,B 0,C 180,E1 -17248.724,E2 -17248.724} C_VEL
LIN {X 0,Y 284.386,Z 253.056,A -85,B 0,C 180,E1 -17252.826,E2 -17252.826} C_VEL
LIN {X 0,Y 284.357,Z 253.064,A -85,B 0,C 180,E1 -17256.706,E2 -17256.706} C_VEL
LIN {X 0,Y 284.393,Z 253.059,A -85,B 0,C 180,E1 -17261.261,E2 -17261.261} C_VEL
LIN {X 0,Y 284.482,Z 253.049,A -85,B 0,C 180,E1 -17264.458,E2 -17264.458} C_VEL
LIN {X 0,Y 284.477,Z 253.049,A -85,B 0,C 180,E1 -17268.601,E2 -17268.601} C_VEL
LIN {X 0,Y 284.65,Z 253.027,A -85,B 0,C 180,E1 -17271.481,E2 -17271.481} C_VEL
LIN {X 0,Y 284.595,Z 253.036,A -85,B 0,C 180,E1 -17274.331,E2 -17274.331} C_VEL
LIN {X 0,Y 284.846,Z 253.004,A -85,B 0,C 180,E1 -17278.586,E2 -17278.586} C_VEL
LIN {X 0,Y 284.844,Z 253.005,A -85,B 0,C 180,E1 -17281.414,E2 -17281.414} C_VEL
LIN {X 0,Y 284.575,Z 253.034,A -85,B 0,C 180,E1 -17283.679,E2 -17283.679} C_VEL
LIN {X 0,Y 283.814,Z 253.131,A -85,B 0,C 180,E1 -17284.86,E2 -17284.86} C_VEL
LIN {X 0,Y 281.013,Z 253.48,A -85,B 0,C 180,E1 -17286.788,E2 -17286.788} C_VEL
LIN {X 0,Y 277.871,Z 253.872,A -85,B 0,C 180,E1 -17289.156,E2 -17289.156} C_VEL
LIN {X 0,Y 277.516,Z 253.916,A -85,B 0,C 180,E1 -17289.973,E2 -17289.973} C_VEL
LIN {X 0,Y 277.423,Z 253.925,A -85,B 0,C 180,E1 -17294.675,E2 -17294.675} C_VEL
LIN {X 0,Y 277.334,Z 253.933,A -85,B 0,C 180,E1 -17299.234,E2 -17299.234} C_VEL
LIN {X 0,Y 277.309,Z 253.942,A -85,B 0,C 180,E1 -17304.171,E2 -17304.171} C_VEL
LIN {X 0,Y 277.318,Z 253.942,A -85,B 0,C 180,E1 -17307.507,E2 -17307.507} C_VEL
LIN {X 0,Y 277.262,Z 253.95,A -85,B 0,C 180,E1 -17310.483,E2 -17310.483} C_VEL
LIN {X 0,Y 277.29,Z 254.004,A -85,B 0,C 180,E1 -17315.212,E2 -17315.212} C_VEL
LIN {X 0,Y 277.772,Z 256.966,A -85,B 0,C 180,E1 -17318.344,E2 -17318.344} C_VEL
LIN {X 0,Y 278.637,Z 261.717,A -85,B 0,C 180,E1 -17322.923,E2 -17322.923} C_VEL
LIN {X 0,Y 279.45,Z 266.114,A -85,B 0,C 180,E1 -17326.831,E2 -17326.831} C_VEL
LIN {X 0,Y 280.215,Z 270.228,A -85,B 0,C 180,E1 -17330.212,E2 -17330.212} C_VEL
LIN {X 0,Y 280.52,Z 273.902,A -85,B 0,C 180,E1 -17333.041,E2 -17333.041} C_VEL
LIN {X 0,Y 279.73,Z 278.075,A -85,B 0,C 180,E1 -17336.007,E2 -17336.007} C_VEL
LIN {X 0,Y 278.42,Z 284.649,A -85,B 0,C 180,E1 -17340.516,E2 -17340.516} C_VEL
LIN {X 0,Y 277.943,Z 287.616,A -85,B 0,C 180,E1 -17342.52,E2 -17342.52} C_VEL
LIN {X 0,Y 279.966,Z 295.863,A -85,B 0,C 180,E1 -17343.115,E2 -17343.115} C_VEL
LIN {X 0,Y 282.598,Z 307.959,A -85,B 0,C 180,E1 -17344.153,E2 -17344.153} C_VEL
LIN {X 0,Y 284.28,Z 319.461,A -85,B 0,C 180,E1 -17345.301,E2 -17345.301} C_VEL
LIN {X 0,Y 285.09,Z 330.223,A -85,B 0,C 180,E1 -17346.547,E2 -17346.547} C_VEL
LIN {X 0,Y 285.205,Z 340.459,A -85,B 0,C 180,E1 -17347.929,E2 -17347.929} C_VEL
LIN {X 0,Y 283.34,Z 350.877,A -85,B 0,C 180,E1 -17349.493,E2 -17349.493} C_VEL
LIN {X 0,Y 281.61,Z 359.409,A -85,B 0,C 180,E1 -17351.071,E2 -17351.071} C_VEL
LIN {X 0,Y 280.095,Z 367.304,A -85,B 0,C 180,E1 -17352.855,E2 -17352.855} C_VEL
LIN {X 0,Y 278.522,Z 375.036,A -85,B 0,C 180,E1 -17355.013,E2 -17355.013} C_VEL
LIN {X 0,Y 276.965,Z 382.177,A -85,B 0,C 180,E1 -17357.546,E2 -17357.546} C_VEL
LIN {X 0,Y 276.181,Z 386.957,A -85,B 0,C 180,E1 -17359.741,E2 -17359.741} C_VEL
LIN {X 0,Y 275.677,Z 390.63,A -85,B 0,C 180,E1 -17361.942,E2 -17361.942} C_VEL
LIN {X 0,Y 275.443,Z 393.481,A -85,B 0,C 180,E1 -17364.325,E2 -17364.325} C_VEL
LIN {X 0,Y 275.404,Z 395.414,A -85,B 0,C 180,E1 -17367.077,E2 -17367.077} C_VEL
LIN {X 0,Y 275.515,Z 395.865,A -85,B 0,C 180,E1 -17370.002,E2 -17370.002} C_VEL
LIN {X 0,Y 275.437,Z 395.494,A -85,B 0,C 180,E1 -17371.464,E2 -17371.464} C_VEL
LIN {X 0,Y 275.423,Z 394.719,A -85,B 0,C 180,E1 -17372.927,E2 -17372.927} C_VEL
LIN {X 0,Y 275.444,Z 393.496,A -85,B 0,C 180,E1 -17374.392,E2 -17374.392} C_VEL
LIN {X 0,Y 275.516,Z 390.886,A -85,B 0,C 180,E1 -17376.594,E2 -17376.594} C_VEL
LIN {X 0,Y 275.832,Z 387.251,A -85,B 0,C 180,E1 -17378.796,E2 -17378.796} C_VEL
LIN {X 0,Y 276.386,Z 382.492,A -85,B 0,C 180,E1 -17380.996,E2 -17380.996} C_VEL
LIN {X 0,Y 277.505,Z 375.343,A -85,B 0,C 180,E1 -17383.55,E2 -17383.55} C_VEL
LIN {X 0,Y 278.789,Z 367.59,A -85,B 0,C 180,E1 -17385.726,E2 -17385.726} C_VEL
LIN {X 0,Y 280.067,Z 359.646,A -85,B 0,C 180,E1 -17387.527,E2 -17387.527} C_VEL
LIN {X 0,Y 281.576,Z 349.949,A -85,B 0,C 180,E1 -17389.314,E2 -17389.314} C_VEL
LIN {X 0,Y 283.406,Z 339.221,A -85,B 0,C 180,E1 -17390.886,E2 -17390.886} C_VEL
LIN {X 0,Y 282.898,Z 328.305,A -85,B 0,C 180,E1 -17392.298,E2 -17392.298} C_VEL
LIN {X 0,Y 282.056,Z 316.913,A -85,B 0,C 180,E1 -17393.497,E2 -17393.497} C_VEL
LIN {X 0,Y 280.348,Z 303.846,A -85,B 0,C 180,E1 -17394.613,E2 -17394.613} C_VEL
LIN {X 0,Y 277.793,Z 290.55,A -85,B 0,C 180,E1 -17395.513,E2 -17395.513} C_VEL
LIN {X 0,Y 277.295,Z 288.027,A -85,B 0,C 180,E1 -17395.65,E2 -17395.65} C_VEL
LIN {X 0,Y 278.438,Z 280.937,A -85,B 0,C 180,E1 -17400.321,E2 -17400.321} C_VEL
LIN {X 0,Y 279.547,Z 274.649,A -85,B 0,C 180,E1 -17404.525,E2 -17404.525} C_VEL
LIN {X 0,Y 280.034,Z 271.038,A -85,B 0,C 180,E1 -17407.039,E2 -17407.039} C_VEL
LIN {X 0,Y 279.688,Z 267.247,A -85,B 0,C 180,E1 -17409.851,E2 -17409.851} C_VEL
LIN {X 0,Y 278.917,Z 263.133,A -85,B 0,C 180,E1 -17413.053,E2 -17413.053} C_VEL
LIN {X 0,Y 278.021,Z 258.271,A -85,B 0,C 180,E1 -17417.148,E2 -17417.148} C_VEL
LIN {X 0,Y 277.302,Z 253.945,A -85,B 0,C 180,E1 -17421.072,E2 -17421.072} C_VEL
LIN {X 0,Y 277.291,Z 253.946,A -85,B 0,C 180,E1 -17424.342,E2 -17424.342} C_VEL
LIN {X 0,Y 277.248,Z 253.949,A -85,B 0,C 180,E1 -17427.837,E2 -17427.837} C_VEL
LIN {X 0,Y 277.253,Z 253.947,A -85,B 0,C 180,E1 -17431.208,E2 -17431.208} C_VEL
LIN {X 0,Y 277.285,Z 253.946,A -85,B 0,C 180,E1 -17434.477,E2 -17434.477} C_VEL
LIN {X 0,Y 277.272,Z 253.946,A -85,B 0,C 180,E1 -17437.654,E2 -17437.654} C_VEL
LIN {X 0,Y 277.31,Z 253.941,A -85,B 0,C 180,E1 -17440.764,E2 -17440.764} C_VEL
LIN {X 0,Y 277.384,Z 253.932,A -85,B 0,C 180,E1 -17445.323,E2 -17445.323} C_VEL
LIN {X 0,Y 277.461,Z 253.926,A -85,B 0,C 180,E1 -17449.787,E2 -17449.787} C_VEL
LIN {X 0,Y 277.636,Z 253.898,A -85,B 0,C 180,E1 -17452.729,E2 -17452.729} C_VEL
LIN {X 0,Y 277.828,Z 253.876,A -85,B 0,C 180,E1 -17458.551,E2 -17458.551} C_VEL
LIN {X 0,Y 277.821,Z 253.878,A -85,B 0,C 180,E1 -17461.45,E2 -17461.45} C_VEL
LIN {X 0,Y 277.607,Z 253.907,A -85,B 0,C 180,E1 -17467.272,E2 -17467.272} C_VEL
LIN {X 0,Y 277.466,Z 253.918,A -85,B 0,C 180,E1 -17470.213,E2 -17470.213} C_VEL
LIN {X 0,Y 277.418,Z 253.926,A -85,B 0,C 180,E1 -17474.675,E2 -17474.675} C_VEL
LIN {X 0,Y 277.326,Z 253.938,A -85,B 0,C 180,E1 -17479.235,E2 -17479.235} C_VEL
LIN {X 0,Y 277.263,Z 253.944,A -85,B 0,C 180,E1 -17483.927,E2 -17483.927} C_VEL
LIN {X 0,Y 277.247,Z 253.948,A -85,B 0,C 180,E1 -17487.47,E2 -17487.47} C_VEL
LIN {X 0,Y 277.236,Z 253.951,A -85,B 0,C 180,E1 -17490.465,E2 -17490.465} C_VEL
LIN {X 0,Y 277.255,Z 253.946,A -85,B 0,C 180,E1 -17493.895,E2 -17493.895} C_VEL
LIN {X 0,Y 277.276,Z 253.944,A -85,B 0,C 180,E1 -17497.468,E2 -17497.468} C_VEL
LIN {X 0,Y 277.218,Z 253.952,A -85,B 0,C 180,E1 -17501.236,E2 -17501.236} C_VEL
LIN {X 0,Y 277.202,Z 253.953,A -85,B 0,C 180,E1 -17505.227,E2 -17505.227} C_VEL
LIN {X 0,Y 277.183,Z 253.957,A -85,B 0,C 180,E1 -17508.756,E2 -17508.756} C_VEL
LIN {X 0,Y 277.238,Z 253.951,A -85,B 0,C 180,E1 -17512.524,E2 -17512.524} C_VEL
LIN {X 0,Y 277.199,Z 253.955,A -85,B 0,C 180,E1 -17516.095,E2 -17516.095} C_VEL
LIN {X 0,Y 277.038,Z 253.973,A -85,B 0,C 180,E1 -17519.602,E2 -17519.602} C_VEL
LIN {X 0,Y 276.837,Z 253.997,A -85,B 0,C 180,E1 -17521.159,E2 -17521.159} C_VEL
LIN {X 0,Y 276.696,Z 256.144,A -85,B 0,C 180,E1 -17524.416,E2 -17524.416} C_VEL
LIN {X 0,Y 276.506,Z 259.524,A -85,B 0,C 180,E1 -17528.671,E2 -17528.671} C_VEL
LIN {X 0,Y 281.165,Z 274.053,A -85,B 0,C 180,E1 -17529.878,E2 -17529.878} C_VEL
LIN {X 0,Y 284.185,Z 286.351,A -85,B 0,C 180,E1 -17531.103,E2 -17531.103} C_VEL
LIN {X 0,Y 285.931,Z 295.627,A -85,B 0,C 180,E1 -17532.192,E2 -17532.192} C_VEL
LIN {X 0,Y 284.586,Z 306.754,A -85,B 0,C 180,E1 -17533.499,E2 -17533.499} C_VEL
LIN {X 0,Y 283.151,Z 317.326,A -85,B 0,C 180,E1 -17535.075,E2 -17535.075} C_VEL
LIN {X 0,Y 281.386,Z 327.738,A -85,B 0,C 180,E1 -17537.008,E2 -17537.008} C_VEL
LIN {X 0,Y 280.1,Z 335.388,A -85,B 0,C 180,E1 -17538.785,E2 -17538.785} C_VEL
LIN {X 0,Y 278.763,Z 342.872,A -85,B 0,C 180,E1 -17540.932,E2 -17540.932} C_VEL
LIN {X 0,Y 277.893,Z 347.996,A -85,B 0,C 180,E1 -17542.733,E2 -17542.733} C_VEL
LIN {X 0,Y 276.902,Z 352.973,A -85,B 0,C 180,E1 -17544.901,E2 -17544.901} C_VEL
LIN {X 0,Y 276.287,Z 356.827,A -85,B 0,C 180,E1 -17547.082,E2 -17547.082} C_VEL
LIN {X 0,Y 276.014,Z 358.811,A -85,B 0,C 180,E1 -17548.539,E2 -17548.539} C_VEL
LIN {X 0,Y 275.818,Z 360.39,A -85,B 0,C 180,E1 -17549.998,E2 -17549.998} C_VEL
LIN {X 0,Y 275.677,Z 361.573,A -85,B 0,C 180,E1 -17551.459,E2 -17551.459} C_VEL
LIN {X 0,Y 275.696,Z 362.681,A -85,B 0,C 180,E1 -17554.384,E2 -17554.384} C_VEL
LIN {X 0,Y 275.831,Z 362.558,A -85,B 0,C 180,E1 -17556.434,E2 -17556.434} C_VEL
LIN {X 0,Y 276.037,Z 361.466,A -85,B 0,C 180,E1 -17558.785,E2 -17558.785} C_VEL
LIN {X 0,Y 276.707,Z 358.629,A -85,B 0,C 180,E1 -17561.721,E2 -17561.721} C_VEL
LIN {X 0,Y 277.526,Z 355.358,A -85,B 0,C 180,E1 -17563.918,E2 -17563.918} C_VEL
LIN {X 0,Y 278.583,Z 351.011,A -85,B 0,C 180,E1 -17566.109,E2 -17566.109} C_VEL
LIN {X 0,Y 279.968,Z 345.457,A -85,B 0,C 180,E1 -17568.285,E2 -17568.285} C_VEL
LIN {X 0,Y 281.705,Z 338.481,A -85,B 0,C 180,E1 -17570.44,E2 -17570.44} C_VEL
LIN {X 0,Y 283.679,Z 329.72,A -85,B 0,C 180,E1 -17572.58,E2 -17572.58} C_VEL
LIN {X 0,Y 285.643,Z 319.793,A -85,B 0,C 180,E1 -17574.518,E2 -17574.518} C_VEL
LIN {X 0,Y 287.587,Z 309.476,A -85,B 0,C 180,E1 -17576.094,E2 -17576.094} C_VEL
LIN {X 0,Y 288.958,Z 301.226,A -85,B 0,C 180,E1 -17577.129,E2 -17577.129} C_VEL
LIN {X 0,Y 287.022,Z 290.726,A -85,B 0,C 180,E1 -17578.546,E2 -17578.546} C_VEL
LIN {X 0,Y 283.878,Z 278.999,A -85,B 0,C 180,E1 -17579.945,E2 -17579.945} C_VEL
LIN {X 0,Y 279.297,Z 266.254,A -85,B 0,C 180,E1 -17581.301,E2 -17581.301} C_VEL
LIN {X 0,Y 277.051,Z 260.715,A -85,B 0,C 180,E1 -17581.828,E2 -17581.828} C_VEL
LIN {X 0,Y 276.946,Z 260.06,A -85,B 0,C 180,E1 -17581.889,E2 -17581.889} C_VEL
LIN {X 0,Y 277.134,Z 257.232,A -85,B 0,C 180,E1 -17585.756,E2 -17585.756} C_VEL
LIN {X 0,Y 277.194,Z 254.766,A -85,B 0,C 180,E1 -17589.332,E2 -17589.332} C_VEL
LIN {X 0,Y 277.147,Z 254.031,A -85,B 0,C 180,E1 -17590.469,E2 -17590.469} C_VEL
LIN {X 0,Y 277.182,Z 253.959,A -85,B 0,C 180,E1 -17593.2,E2 -17593.2} C_VEL
LIN {X 0,Y 277.208,Z 253.955,A -85,B 0,C 180,E1 -17597.323,E2 -17597.323} C_VEL
LIN {X 0,Y 277.267,Z 253.947,A -85,B 0,C 180,E1 -17601.788,E2 -17601.788} C_VEL
LIN {X 0,Y 277.295,Z 253.945,A -85,B 0,C 180,E1 -17604.343,E2 -17604.343} C_VEL
LIN {X 0,Y 277.235,Z 253.952,A -85,B 0,C 180,E1 -17607.835,E2 -17607.835} C_VEL
LIN {X 0,Y 277.277,Z 253.946,A -85,B 0,C 180,E1 -17611.211,E2 -17611.211} C_VEL
LIN {X 0,Y 277.303,Z 253.944,A -85,B 0,C 180,E1 -17614.478,E2 -17614.478} C_VEL
LIN {X 0,Y 277.276,Z 253.947,A -85,B 0,C 180,E1 -17617.654,E2 -17617.654} C_VEL
LIN {X 0,Y 277.335,Z 253.941,A -85,B 0,C 180,E1 -17620.765,E2 -17620.765} C_VEL
LIN {X 0,Y 277.424,Z 253.929,A -85,B 0,C 180,E1 -17625.325,E2 -17625.325} C_VEL
LIN {X 0,Y 277.496,Z 253.919,A -85,B 0,C 180,E1 -17629.788,E2 -17629.788} C_VEL
LIN {X 0,Y 277.645,Z 253.9,A -85,B 0,C 180,E1 -17632.729,E2 -17632.729} C_VEL
LIN {X 0,Y 277.813,Z 253.88,A -85,B 0,C 180,E1 -17638.55,E2 -17638.55} C_VEL
LIN {X 0,Y 277.81,Z 253.881,A -85,B 0,C 180,E1 -17641.449,E2 -17641.449} C_VEL
LIN {X 0,Y 277.644,Z 253.902,A -85,B 0,C 180,E1 -17647.271,E2 -17647.271} C_VEL
LIN {X 0,Y 277.516,Z 253.916,A -85,B 0,C 180,E1 -17649.973,E2 -17649.973} C_VEL
LIN {X 0,Y 276.772,Z 254.011,A -85,B 0,C 180,E1 -17651.182,E2 -17651.182} C_VEL
LIN {X 0,Y 273.885,Z 254.366,A -85,B 0,C 180,E1 -17653.153,E2 -17653.153} C_VEL
LIN {X 0,Y 271.474,Z 254.665,A -85,B 0,C 180,E1 -17654.754,E2 -17654.754} C_VEL
LIN {X 0,Y 270.436,Z 254.792,A -85,B 0,C 180,E1 -17655.995,E2 -17655.995} C_VEL
LIN {X 0,Y 270.347,Z 254.804,A -85,B 0,C 180,E1 -17656.416,E2 -17656.416} C_VEL
LIN {X 0,Y 270.282,Z 254.819,A -85,B 0,C 180,E1 -17660.602,E2 -17660.602} C_VEL
LIN {X 0,Y 270.264,Z 254.819,A -85,B 0,C 180,E1 -17664.586,E2 -17664.586} C_VEL
LIN {X 0,Y 270.263,Z 254.821,A -85,B 0,C 180,E1 -17667.91,E2 -17667.91} C_VEL
LIN {X 0,Y 270.175,Z 254.831,A -85,B 0,C 180,E1 -17671.349,E2 -17671.349} C_VEL
LIN {X 0,Y 270.22,Z 254.913,A -85,B 0,C 180,E1 -17674.385,E2 -17674.385} C_VEL
LIN {X 0,Y 270.879,Z 258.681,A -85,B 0,C 180,E1 -17678.512,E2 -17678.512} C_VEL
LIN {X 0,Y 271.579,Z 262.455,A -85,B 0,C 180,E1 -17682.286,E2 -17682.286} C_VEL
LIN {X 0,Y 272.373,Z 266.813,A -85,B 0,C 180,E1 -17686.26,E2 -17686.26} C_VEL
LIN {X 0,Y 273.27,Z 271.798,A -85,B 0,C 180,E1 -17690.493,E2 -17690.493} C_VEL
LIN {X 0,Y 273.496,Z 274.721,A -85,B 0,C 180,E1 -17692.807,E2 -17692.807} C_VEL
LIN {X 0,Y 272.808,Z 278.419,A -85,B 0,C 180,E1 -17695.525,E2 -17695.525} C_VEL
LIN {X 0,Y 271.56,Z 284.298,A -85,B 0,C 180,E1 -17699.694,E2 -17699.694} C_VEL
LIN {X 0,Y 271.057,Z 287.174,A -85,B 0,C 180,E1 -17701.704,E2 -17701.704} C_VEL
LIN {X 0,Y 273.899,Z 298.517,A -85,B 0,C 180,E1 -17702.592,E2 -17702.592} C_VEL
LIN {X 0,Y 276.345,Z 310.447,A -85,B 0,C 180,E1 -17703.699,E2 -17703.699} C_VEL
LIN {X 0,Y 277.794,Z 321.33,A -85,B 0,C 180,E1 -17704.864,E2 -17704.864} C_VEL
LIN {X 0,Y 278.466,Z 332.051,A -85,B 0,C 180,E1 -17706.186,E2 -17706.186} C_VEL
LIN {X 0,Y 278.288,Z 342.879,A -85,B 0,C 180,E1 -17707.742,E2 -17707.742} C_VEL
LIN {X 0,Y 276.037,Z 353.695,A -85,B 0,C 180,E1 -17709.51,E2 -17709.51} C_VEL
LIN {X 0,Y 274.113,Z 362.83,A -85,B 0,C 180,E1 -17711.387,E2 -17711.387} C_VEL
LIN {X 0,Y 272.36,Z 371.108,A -85,B 0,C 180,E1 -17713.513,E2 -17713.513} C_VEL
LIN {X 0,Y 270.86,Z 378.016,A -85,B 0,C 180,E1 -17715.732,E2 -17715.732} C_VEL
LIN {X 0,Y 269.666,Z 383.566,A -85,B 0,C 180,E1 -17717.968,E2 -17717.968} C_VEL
LIN {X 0,Y 268.945,Z 387.942,A -85,B 0,C 180,E1 -17720.223,E2 -17720.223} C_VEL
LIN {X 0,Y 268.523,Z 391.256,A -85,B 0,C 180,E1 -17722.483,E2 -17722.483} C_VEL
LIN {X 0,Y 268.351,Z 393.306,A -85,B 0,C 180,E1 -17724.388,E2 -17724.388} C_VEL
LIN {X 0,Y 268.333,Z 395.002,A -85,B 0,C 180,E1 -17727,E2 -17727} C_VEL
LIN {X 0,Y 268.427,Z 395.433,A -85,B 0,C 180,E1 -17730.002,E2 -17730.002} C_VEL
LIN {X 0,Y 268.355,Z 395.052,A -85,B 0,C 180,E1 -17731.503,E2 -17731.503} C_VEL
LIN {X 0,Y 268.352,Z 394.258,A -85,B 0,C 180,E1 -17733.005,E2 -17733.005} C_VEL
LIN {X 0,Y 268.392,Z 391.754,A -85,B 0,C 180,E1 -17735.7,E2 -17735.7} C_VEL
LIN {X 0,Y 268.637,Z 388.061,A -85,B 0,C 180,E1 -17738.275,E2 -17738.275} C_VEL
LIN {X 0,Y 269.165,Z 383.667,A -85,B 0,C 180,E1 -17740.533,E2 -17740.533} C_VEL
LIN {X 0,Y 269.963,Z 378.069,A -85,B 0,C 180,E1 -17742.787,E2 -17742.787} C_VEL
LIN {X 0,Y 271.188,Z 371.091,A -85,B 0,C 180,E1 -17745.022,E2 -17745.022} C_VEL
LIN {X 0,Y 272.597,Z 363.114,A -85,B 0,C 180,E1 -17747.07,E2 -17747.07} C_VEL
LIN {X 0,Y 274.175,Z 353.38,A -85,B 0,C 180,E1 -17749.078,E2 -17749.078} C_VEL
LIN {X 0,Y 275.863,Z 343.549,A -85,B 0,C 180,E1 -17750.703,E2 -17750.703} C_VEL
LIN {X 0,Y 276.512,Z 338.433,A -85,B 0,C 180,E1 -17751.432,E2 -17751.432} C_VEL
LIN {X 0,Y 276.016,Z 328.111,A -85,B 0,C 180,E1 -17752.802,E2 -17752.802} C_VEL
LIN {X 0,Y 275.139,Z 315.835,A -85,B 0,C 180,E1 -17754.125,E2 -17754.125} C_VEL
LIN {X 0,Y 273.302,Z 302.324,A -85,B 0,C 180,E1 -17755.304,E2 -17755.304} C_VEL
LIN {X 0,Y 270.664,Z 289.59,A -85,B 0,C 180,E1 -17756.197,E2 -17756.197} C_VEL
LIN {X 0,Y 270.382,Z 287.526,A -85,B 0,C 180,E1 -17756.33,E2 -17756.33} C_VEL
LIN {X 0,Y 271.353,Z 281.671,A -85,B 0,C 180,E1 -17760.337,E2 -17760.337} C_VEL
LIN {X 0,Y 272.49,Z 275.513,A -85,B 0,C 180,E1 -17764.573,E2 -17764.573} C_VEL
LIN {X 0,Y 273.008,Z 272.038,A -85,B 0,C 180,E1 -17767.058,E2 -17767.058} C_VEL
LIN {X 0,Y 272.62,Z 268.015,A -85,B 0,C 180,E1 -17770.13,E2 -17770.13} C_VEL
LIN {X 0,Y 271.803,Z 263.678,A -85,B 0,C 180,E1 -17773.615,E2 -17773.615} C_VEL
LIN {X 0,Y 270.944,Z 259.128,A -85,B 0,C 180,E1 -17777.591,E2 -17777.591} C_VEL
LIN {X 0,Y 270.255,Z 254.823,A -85,B 0,C 180,E1 -17781.65,E2 -17781.65} C_VEL
LIN {X 0,Y 270.209,Z 254.827,A -85,B 0,C 180,E1 -17785.096,E2 -17785.096} C_VEL
LIN {X 0,Y 270.192,Z 254.827,A -85,B 0,C 180,E1 -17789.137,E2 -17789.137} C_VEL
LIN {X 0,Y 270.229,Z 254.824,A -85,B 0,C 180,E1 -17792.164,E2 -17792.164} C_VEL
LIN {X 0,Y 270.239,Z 254.821,A -85,B 0,C 180,E1 -17795.542,E2 -17795.542} C_VEL
LIN {X 0,Y 270.258,Z 254.822,A -85,B 0,C 180,E1 -17800.241,E2 -17800.241} C_VEL
LIN {X 0,Y 270.354,Z 254.808,A -85,B 0,C 180,E1 -17804.933,E2 -17804.933} C_VEL
LIN {X 0,Y 270.393,Z 254.805,A -85,B 0,C 180,E1 -17809.517,E2 -17809.517} C_VEL
LIN {X 0,Y 270.593,Z 254.776,A -85,B 0,C 180,E1 -17812.538,E2 -17812.538} C_VEL
LIN {X 0,Y 270.794,Z 254.752,A -85,B 0,C 180,E1 -17818.513,E2 -17818.513} C_VEL
LIN {X 0,Y 270.785,Z 254.755,A -85,B 0,C 180,E1 -17821.487,E2 -17821.487} C_VEL
LIN {X 0,Y 270.569,Z 254.783,A -85,B 0,C 180,E1 -17827.463,E2 -17827.463} C_VEL
LIN {X 0,Y 270.419,Z 254.797,A -85,B 0,C 180,E1 -17830.482,E2 -17830.482} C_VEL
LIN {X 0,Y 270.377,Z 254.804,A -85,B 0,C 180,E1 -17835.066,E2 -17835.066} C_VEL
LIN {X 0,Y 270.266,Z 254.815,A -85,B 0,C 180,E1 -17839.759,E2 -17839.759} C_VEL
LIN {X 0,Y 270.185,Z 254.828,A -85,B 0,C 180,E1 -17844.595,E2 -17844.595} C_VEL
LIN {X 0,Y 270.194,Z 254.826,A -85,B 0,C 180,E1 -17847.918,E2 -17847.918} C_VEL
LIN {X 0,Y 270.177,Z 254.829,A -85,B 0,C 180,E1 -17851.35,E2 -17851.35} C_VEL
LIN {X 0,Y 270.21,Z 254.826,A -85,B 0,C 180,E1 -17854.905,E2 -17854.905} C_VEL
LIN {X 0,Y 270.206,Z 254.827,A -85,B 0,C 180,E1 -17858.709,E2 -17858.709} C_VEL
LIN {X 0,Y 270.173,Z 254.829,A -85,B 0,C 180,E1 -17863.248,E2 -17863.248} C_VEL
LIN {X 0,Y 270.158,Z 254.832,A -85,B 0,C 180,E1 -17867.436,E2 -17867.436} C_VEL
LIN {X 0,Y 270.158,Z 254.832,A -85,B 0,C 180,E1 -17871.363,E2 -17871.363} C_VEL
LIN {X 0,Y 270.18,Z 254.829,A -85,B 0,C 180,E1 -17875.089,E2 -17875.089} C_VEL
LIN {X 0,Y 270.023,Z 254.844,A -85,B 0,C 180,E1 -17878.629,E2 -17878.629} C_VEL
LIN {X 0,Y 269.87,Z 254.865,A -85,B 0,C 180,E1 -17880.341,E2 -17880.341} C_VEL
LIN {X 0,Y 269.753,Z 255.623,A -85,B 0,C 180,E1 -17882.353,E2 -17882.353} C_VEL
LIN {X 0,Y 269.595,Z 258.254,A -85,B 0,C 180,E1 -17885.841,E2 -17885.841} C_VEL
LIN {X 0,Y 269.511,Z 260.178,A -85,B 0,C 180,E1 -17888.039,E2 -17888.039} C_VEL
LIN {X 0,Y 273.818,Z 273.238,A -85,B 0,C 180,E1 -17889.152,E2 -17889.152} C_VEL
LIN {X 0,Y 276.844,Z 284.785,A -85,B 0,C 180,E1 -17890.325,E2 -17890.325} C_VEL
LIN {X 0,Y 279.159,Z 296.649,A -85,B 0,C 180,E1 -17891.745,E2 -17891.745} C_VEL
LIN {X 0,Y 277.843,Z 307.616,A -85,B 0,C 180,E1 -17893.087,E2 -17893.087} C_VEL
LIN {X 0,Y 276.351,Z 318.113,A -85,B 0,C 180,E1 -17894.699,E2 -17894.699} C_VEL
LIN {X 0,Y 274.523,Z 328.445,A -85,B 0,C 180,E1 -17896.677,E2 -17896.677} C_VEL
LIN {X 0,Y 273.19,Z 336.043,A -85,B 0,C 180,E1 -17898.498,E2 -17898.498} C_VEL
LIN {X 0,Y 271.778,Z 343.488,A -85,B 0,C 180,E1 -17900.697,E2 -17900.697} C_VEL
LIN {X 0,Y 270.874,Z 348.576,A -85,B 0,C 180,E1 -17902.544,E2 -17902.544} C_VEL
LIN {X 0,Y 269.875,Z 353.519,A -85,B 0,C 180,E1 -17904.768,E2 -17904.768} C_VEL
LIN {X 0,Y 269.225,Z 357.343,A -85,B 0,C 180,E1 -17907.005,E2 -17907.005} C_VEL
LIN {X 0,Y 268.945,Z 359.313,A -85,B 0,C 180,E1 -17908.5,E2 -17908.5} C_VEL
LIN {X 0,Y 268.729,Z 360.878,A -85,B 0,C 180,E1 -17909.998,E2 -17909.998} C_VEL
LIN {X 0,Y 268.585,Z 362.04,A -85,B 0,C 180,E1 -17911.497,E2 -17911.497} C_VEL
LIN {X 0,Y 268.637,Z 363.114,A -85,B 0,C 180,E1 -17914.499,E2 -17914.499} C_VEL
LIN {X 0,Y 268.75,Z 363.023,A -85,B 0,C 180,E1 -17916.418,E2 -17916.418} C_VEL
LIN {X 0,Y 268.99,Z 361.847,A -85,B 0,C 180,E1 -17919.017,E2 -17919.017} C_VEL
LIN {X 0,Y 269.716,Z 358.982,A -85,B 0,C 180,E1 -17922.03,E2 -17922.03} C_VEL
LIN {X 0,Y 270.607,Z 355.681,A -85,B 0,C 180,E1 -17924.282,E2 -17924.282} C_VEL
LIN {X 0,Y 271.728,Z 351.302,A -85,B 0,C 180,E1 -17926.527,E2 -17926.527} C_VEL
LIN {X 0,Y 273.471,Z 344.631,A -85,B 0,C 180,E1 -17929.125,E2 -17929.125} C_VEL
LIN {X 0,Y 275.317,Z 337.329,A -85,B 0,C 180,E1 -17931.329,E2 -17931.329} C_VEL
LIN {X 0,Y 277.443,Z 328.232,A -85,B 0,C 180,E1 -17933.511,E2 -17933.511} C_VEL
LIN {X 0,Y 279.378,Z 318.737,A -85,B 0,C 180,E1 -17935.316,E2 -17935.316} C_VEL
LIN {X 0,Y 281.437,Z 308.166,A -85,B 0,C 180,E1 -17936.909,E2 -17936.909} C_VEL
LIN {X 0,Y 282.376,Z 302.613,A -85,B 0,C 180,E1 -17937.614,E2 -17937.614} C_VEL
LIN {X 0,Y 280.438,Z 292.05,A -85,B 0,C 180,E1 -17939.115,E2 -17939.115} C_VEL
LIN {X 0,Y 277.439,Z 280.706,A -85,B 0,C 180,E1 -17940.539,E2 -17940.539} C_VEL
LIN {X 0,Y 272.934,Z 268.233,A -85,B 0,C 180,E1 -17941.951,E2 -17941.951} C_VEL
LIN {X 0,Y 270.043,Z 260.939,A -85,B 0,C 180,E1 -17942.682,E2 -17942.682} C_VEL
LIN {X 0,Y 269.973,Z 260.509,A -85,B 0,C 180,E1 -17942.744,E2 -17942.744} C_VEL
LIN {X 0,Y 270.14,Z 257.679,A -85,B 0,C 180,E1 -17946.75,E2 -17946.75} C_VEL
LIN {X 0,Y 270.217,Z 256.346,A -85,B 0,C 180,E1 -17948.715,E2 -17948.715} C_VEL
LIN {X 0,Y 270.111,Z 254.884,A -85,B 0,C 180,E1 -17951.014,E2 -17951.014} C_VEL
LIN {X 0,Y 270.139,Z 254.837,A -85,B 0,C 180,E1 -17954.62,E2 -17954.62} C_VEL
LIN {X 0,Y 270.165,Z 254.832,A -85,B 0,C 180,E1 -17957.44,E2 -17957.44} C_VEL
LIN {X 0,Y 270.199,Z 254.827,A -85,B 0,C 180,E1 -17961.372,E2 -17961.372} C_VEL
LIN {X 0,Y 270.207,Z 254.827,A -85,B 0,C 180,E1 -17965.095,E2 -17965.095} C_VEL
LIN {X 0,Y 270.191,Z 254.825,A -85,B 0,C 180,E1 -17969.129,E2 -17969.129} C_VEL
LIN {X 0,Y 270.255,Z 254.817,A -85,B 0,C 180,E1 -17972.144,E2 -17972.144} C_VEL
LIN {X 0,Y 270.268,Z 254.819,A -85,B 0,C 180,E1 -17975.518,E2 -17975.518} C_VEL
LIN {X 0,Y 270.291,Z 254.816,A -85,B 0,C 180,E1 -17980.243,E2 -17980.243} C_VEL
LIN {X 0,Y 270.392,Z 254.804,A -85,B 0,C 180,E1 -17984.935,E2 -17984.935} C_VEL
LIN {X 0,Y 270.431,Z 254.8,A -85,B 0,C 180,E1 -17989.518,E2 -17989.518} C_VEL
LIN {X 0,Y 270.603,Z 254.778,A -85,B 0,C 180,E1 -17992.538,E2 -17992.538} C_VEL
LIN {X 0,Y 270.779,Z 254.756,A -85,B 0,C 180,E1 -17998.513,E2 -17998.513} C_VEL
LIN {X 0,Y 270.776,Z 254.757,A -85,B 0,C 180,E1 -18001.487,E2 -18001.487} C_VEL
LIN {X 0,Y 270.602,Z 254.779,A -85,B 0,C 180,E1 -18007.461,E2 -18007.461} C_VEL
LIN {X 0,Y 270.431,Z 254.798,A -85,B 0,C 180,E1 -18010.481,E2 -18010.481} C_VEL
LIN {X 0,Y 270.392,Z 254.798,A -85,B 0,C 180,E1 -18015.065,E2 -18015.065} C_VEL
LIN {X 0,Y 270.347,Z 254.804,A -85,B 0,C 180,E1 -18016.416,E2 -18016.416} C_VEL
LIN {X 0,Y 269.644,Z 254.898,A -85,B 0,C 180,E1 -18017.659,E2 -18017.659} C_VEL
LIN {X 0,Y 266.704,Z 255.265,A -85,B 0,C 180,E1 -18019.684,E2 -18019.684} C_VEL
LIN {X 0,Y 264.238,Z 255.57,A -85,B 0,C 180,E1 -18021.33,E2 -18021.33} C_VEL
LIN {X 0,Y 263.209,Z 255.699,A -85,B 0,C 180,E1 -18022.608,E2 -18022.608} C_VEL
LIN {X 0,Y 263.14,Z 255.706,A -85,B 0,C 180,E1 -18023.041,E2 -18023.041} C_VEL
LIN {X 0,Y 263.199,Z 255.701,A -85,B 0,C 180,E1 -18025.292,E2 -18025.292} C_VEL
LIN {X 0,Y 263.171,Z 255.703,A -85,B 0,C 180,E1 -18028.731,E2 -18028.731} C_VEL
LIN {X 0,Y 263.164,Z 255.734,A -85,B 0,C 180,E1 -18033.422,E2 -18033.422} C_VEL
LIN {X 0,Y 263.7,Z 258.734,A -85,B 0,C 180,E1 -18036.918,E2 -18036.918} C_VEL
LIN {X 0,Y 264.553,Z 263.558,A -85,B 0,C 180,E1 -18041.945,E2 -18041.945} C_VEL
LIN {X 0,Y 265.281,Z 267.475,A -85,B 0,C 180,E1 -18045.668,E2 -18045.668} C_VEL
LIN {X 0,Y 266.181,Z 272.358,A -85,B 0,C 180,E1 -18049.968,E2 -18049.968} C_VEL
LIN {X 0,Y 266.476,Z 275.668,A -85,B 0,C 180,E1 -18052.659,E2 -18052.659} C_VEL
LIN {X 0,Y 265.935,Z 278.755,A -85,B 0,C 180,E1 -18055.01,E2 -18055.01} C_VEL
LIN {X 0,Y 264.508,Z 285.124,A -85,B 0,C 180,E1 -18059.683,E2 -18059.683} C_VEL
LIN {X 0,Y 264.216,Z 286.705,A -85,B 0,C 180,E1 -18060.829,E2 -18060.829} C_VEL
LIN {X 0,Y 267.847,Z 301.213,A -85,B 0,C 180,E1 -18062.061,E2 -18062.061} C_VEL
LIN {X 0,Y 270.326,Z 314.687,A -85,B 0,C 180,E1 -18063.433,E2 -18063.433} C_VEL
LIN {X 0,Y 271.608,Z 327.105,A -85,B 0,C 180,E1 -18064.91,E2 -18064.91} C_VEL
LIN {X 0,Y 271.809,Z 337.673,A -85,B 0,C 180,E1 -18066.376,E2 -18066.376} C_VEL
LIN {X 0,Y 271.467,Z 343.931,A -85,B 0,C 180,E1 -18067.353,E2 -18067.353} C_VEL
LIN {X 0,Y 269.369,Z 353.518,A -85,B 0,C 180,E1 -18068.979,E2 -18068.979} C_VEL
LIN {X 0,Y 267.371,Z 362.611,A -85,B 0,C 180,E1 -18070.9,E2 -18070.9} C_VEL
LIN {X 0,Y 265.545,Z 370.838,A -85,B 0,C 180,E1 -18073.077,E2 -18073.077} C_VEL
LIN {X 0,Y 263.951,Z 377.716,A -85,B 0,C 180,E1 -18075.35,E2 -18075.35} C_VEL
LIN {X 0,Y 262.677,Z 383.239,A -85,B 0,C 180,E1 -18077.643,E2 -18077.643} C_VEL
LIN {X 0,Y 261.904,Z 387.591,A -85,B 0,C 180,E1 -18079.957,E2 -18079.957} C_VEL
LIN {X 0,Y 261.443,Z 390.882,A -85,B 0,C 180,E1 -18082.278,E2 -18082.278} C_VEL
LIN {X 0,Y 261.252,Z 393.102,A -85,B 0,C 180,E1 -18084.472,E2 -18084.472} C_VEL
LIN {X 0,Y 261.263,Z 394.591,A -85,B 0,C 180,E1 -18086.918,E2 -18086.918} C_VEL
LIN {X 0,Y 261.342,Z 395.001,A -85,B 0,C 180,E1 -18090.002,E2 -18090.002} C_VEL
LIN {X 0,Y 261.276,Z 394.611,A -85,B 0,C 180,E1 -18091.544,E2 -18091.544} C_VEL
LIN {X 0,Y 261.283,Z 393.796,A -85,B 0,C 180,E1 -18093.086,E2 -18093.086} C_VEL
LIN {X 0,Y 261.294,Z 391.541,A -85,B 0,C 180,E1 -18095.624,E2 -18095.624} C_VEL
LIN {X 0,Y 261.582,Z 387.552,A -85,B 0,C 180,E1 -18098.5,E2 -18098.5} C_VEL
LIN {X 0,Y 262.127,Z 383.133,A -85,B 0,C 180,E1 -18100.82,E2 -18100.82} C_VEL
LIN {X 0,Y 262.985,Z 377.508,A -85,B 0,C 180,E1 -18103.132,E2 -18103.132} C_VEL
LIN {X 0,Y 264.258,Z 370.496,A -85,B 0,C 180,E1 -18105.426,E2 -18105.426} C_VEL
LIN {X 0,Y 265.608,Z 363.352,A -85,B 0,C 180,E1 -18107.317,E2 -18107.317} C_VEL
LIN {X 0,Y 267.102,Z 354.671,A -85,B 0,C 180,E1 -18109.204,E2 -18109.204} C_VEL
LIN {X 0,Y 268.821,Z 345.186,A -85,B 0,C 180,E1 -18110.87,E2 -18110.87} C_VEL
LIN {X 0,Y 269.664,Z 340.297,A -85,B 0,C 180,E1 -18111.602,E2 -18111.602} C_VEL
LIN {X 0,Y 269.206,Z 328.659,A -85,B 0,C 180,E1 -18113.235,E2 -18113.235} C_VEL
LIN {X 0,Y 268.418,Z 316.58,A -85,B 0,C 180,E1 -18114.608,E2 -18114.608} C_VEL
LIN {X 0,Y 266.607,Z 303.142,A -85,B 0,C 180,E1 -18115.845,E2 -18115.845} C_VEL
LIN {X 0,Y 263.907,Z 289.661,A -85,B 0,C 180,E1 -18116.839,E2 -18116.839} C_VEL
LIN {X 0,Y 263.436,Z 287.119,A -85,B 0,C 180,E1 -18117.026,E2 -18117.026} C_VEL
LIN {X 0,Y 264.474,Z 281.351,A -85,B 0,C 180,E1 -18121.081,E2 -18121.081} C_VEL
LIN {X 0,Y 265.711,Z 275.041,A -85,B 0,C 180,E1 -18125.586,E2 -18125.586} C_VEL
LIN {X 0,Y 265.925,Z 271.293,A -85,B 0,C 180,E1 -18128.396,E2 -18128.396} C_VEL
LIN {X 0,Y 265.191,Z 266.735,A -85,B 0,C 180,E1 -18132.094,E2 -18132.094} C_VEL
LIN {X 0,Y 264.263,Z 261.955,A -85,B 0,C 180,E1 -18136.254,E2 -18136.254} C_VEL
LIN {X 0,Y 263.462,Z 257.256,A -85,B 0,C 180,E1 -18140.681,E2 -18140.681} C_VEL
LIN {X 0,Y 263.189,Z 255.703,A -85,B 0,C 180,E1 -18142.426,E2 -18142.426} C_VEL
LIN {X 0,Y 263.159,Z 255.705,A -85,B 0,C 180,E1 -18145.887,E2 -18145.887} C_VEL
LIN {X 0,Y 263.134,Z 255.706,A -85,B 0,C 180,E1 -18149.505,E2 -18149.505} C_VEL
LIN {X 0,Y 263.154,Z 255.704,A -85,B 0,C 180,E1 -18152.998,E2 -18152.998} C_VEL
LIN {X 0,Y 263.157,Z 255.706,A -85,B 0,C 180,E1 -18156.385,E2 -18156.385} C_VEL
LIN {X 0,Y 263.243,Z 255.694,A -85,B 0,C 180,E1 -18159.692,E2 -18159.692} C_VEL
LIN {X 0,Y 263.304,Z 255.687,A -85,B 0,C 180,E1 -18164.519,E2 -18164.519} C_VEL
LIN {X 0,Y 263.338,Z 255.683,A -85,B 0,C 180,E1 -18169.233,E2 -18169.233} C_VEL
LIN {X 0,Y 263.553,Z 255.654,A -85,B 0,C 180,E1 -18172.338,E2 -18172.338} C_VEL
LIN {X 0,Y 263.758,Z 255.628,A -85,B 0,C 180,E1 -18178.473,E2 -18178.473} C_VEL
LIN {X 0,Y 263.749,Z 255.632,A -85,B 0,C 180,E1 -18181.527,E2 -18181.527} C_VEL
LIN {X 0,Y 263.534,Z 255.658,A -85,B 0,C 180,E1 -18187.663,E2 -18187.663} C_VEL
LIN {X 0,Y 263.358,Z 255.677,A -85,B 0,C 180,E1 -18190.766,E2 -18190.766} C_VEL
LIN {X 0,Y 263.319,Z 255.684,A -85,B 0,C 180,E1 -18195.48,E2 -18195.48} C_VEL
LIN {X 0,Y 263.245,Z 255.69,A -85,B 0,C 180,E1 -18200.308,E2 -18200.308} C_VEL
LIN {X 0,Y 263.129,Z 255.707,A -85,B 0,C 180,E1 -18205.3,E2 -18205.3} C_VEL
LIN {X 0,Y 263.127,Z 255.708,A -85,B 0,C 180,E1 -18208.736,E2 -18208.736} C_VEL
LIN {X 0,Y 263.134,Z 255.708,A -85,B 0,C 180,E1 -18212.288,E2 -18212.288} C_VEL
LIN {X 0,Y 263.191,Z 255.7,A -85,B 0,C 180,E1 -18216.762,E2 -18216.762} C_VEL
LIN {X 0,Y 263.132,Z 255.707,A -85,B 0,C 180,E1 -18221.592,E2 -18221.592} C_VEL
LIN {X 0,Y 263.105,Z 255.712,A -85,B 0,C 180,E1 -18226.009,E2 -18226.009} C_VEL
LIN {X 0,Y 263.079,Z 255.716,A -85,B 0,C 180,E1 -18230.12,E2 -18230.12} C_VEL
LIN {X 0,Y 263.152,Z 255.708,A -85,B 0,C 180,E1 -18234.014,E2 -18234.014} C_VEL
LIN {X 0,Y 263.034,Z 255.718,A -85,B 0,C 180,E1 -18237.696,E2 -18237.696} C_VEL
LIN {X 0,Y 262.714,Z 255.857,A -85,B 0,C 180,E1 -18241.212,E2 -18241.212} C_VEL
LIN {X 0,Y 262.59,Z 258.359,A -85,B 0,C 180,E1 -18244.643,E2 -18244.643} C_VEL
LIN {X 0,Y 262.476,Z 260.369,A -85,B 0,C 180,E1 -18247.308,E2 -18247.308} C_VEL
LIN {X 0,Y 267.419,Z 275.326,A -85,B 0,C 180,E1 -18248.675,E2 -18248.675} C_VEL
LIN {X 0,Y 270.418,Z 287.158,A -85,B 0,C 180,E1 -18249.951,E2 -18249.951} C_VEL
LIN {X 0,Y 272.401,Z 297.653,A -85,B 0,C 180,E1 -18251.278,E2 -18251.278} C_VEL
LIN {X 0,Y 271.919,Z 303.009,A -85,B 0,C 180,E1 -18251.93,E2 -18251.93} C_VEL
LIN {X 0,Y 270.441,Z 313.384,A -85,B 0,C 180,E1 -18253.388,E2 -18253.388} C_VEL
LIN {X 0,Y 268.658,Z 323.859,A -85,B 0,C 180,E1 -18255.221,E2 -18255.221} C_VEL
LIN {X 0,Y 267.178,Z 332.006,A -85,B 0,C 180,E1 -18256.993,E2 -18256.993} C_VEL
LIN {X 0,Y 265.473,Z 340.602,A -85,B 0,C 180,E1 -18259.318,E2 -18259.318} C_VEL
LIN {X 0,Y 264.291,Z 347.236,A -85,B 0,C 180,E1 -18261.588,E2 -18261.588} C_VEL
LIN {X 0,Y 263.106,Z 352.559,A -85,B 0,C 180,E1 -18263.864,E2 -18263.864} C_VEL
LIN {X 0,Y 262.361,Z 356.708,A -85,B 0,C 180,E1 -18266.158,E2 -18266.158} C_VEL
LIN {X 0,Y 261.862,Z 359.816,A -85,B 0,C 180,E1 -18268.46,E2 -18268.46} C_VEL
LIN {X 0,Y 261.64,Z 361.367,A -85,B 0,C 180,E1 -18269.998,E2 -18269.998} C_VEL
LIN {X 0,Y 261.495,Z 362.503,A -85,B 0,C 180,E1 -18271.538,E2 -18271.538} C_VEL
LIN {X 0,Y 261.556,Z 363.548,A -85,B 0,C 180,E1 -18274.621,E2 -18274.621} C_VEL
LIN {X 0,Y 261.686,Z 363.473,A -85,B 0,C 180,E1 -18276.434,E2 -18276.434} C_VEL
LIN {X 0,Y 261.964,Z 362.227,A -85,B 0,C 180,E1 -18279.261,E2 -18279.261} C_VEL
LIN {X 0,Y 262.745,Z 359.335,A -85,B 0,C 180,E1 -18282.354,E2 -18282.354} C_VEL
LIN {X 0,Y 263.703,Z 356.004,A -85,B 0,C 180,E1 -18284.664,E2 -18284.664} C_VEL
LIN {X 0,Y 265.21,Z 350.503,A -85,B 0,C 180,E1 -18287.446,E2 -18287.446} C_VEL
LIN {X 0,Y 267.046,Z 343.758,A -85,B 0,C 180,E1 -18290.004,E2 -18290.004} C_VEL
LIN {X 0,Y 269.04,Z 336.166,A -85,B 0,C 180,E1 -18292.255,E2 -18292.255} C_VEL
LIN {X 0,Y 270.921,Z 328.36,A -85,B 0,C 180,E1 -18294.113,E2 -18294.113} C_VEL
LIN {X 0,Y 272.942,Z 318.8,A -85,B 0,C 180,E1 -18295.957,E2 -18295.957} C_VEL
LIN {X 0,Y 275.068,Z 308.295,A -85,B 0,C 180,E1 -18297.562,E2 -18297.562} C_VEL
LIN {X 0,Y 275.703,Z 303.33,A -85,B 0,C 180,E1 -18298.229,E2 -18298.229} C_VEL
LIN {X 0,Y 273.893,Z 293.5,A -85,B 0,C 180,E1 -18299.688,E2 -18299.688} C_VEL
LIN {X 0,Y 271.004,Z 282.531,A -85,B 0,C 180,E1 -18301.151,E2 -18301.151} C_VEL
LIN {X 0,Y 266.638,Z 270.206,A -85,B 0,C 180,E1 -18302.628,E2 -18302.628} C_VEL
LIN {X 0,Y 263.089,Z 261.513,A -85,B 0,C 180,E1 -18303.566,E2 -18303.566} C_VEL
LIN {X 0,Y 263.024,Z 260.959,A -85,B 0,C 180,E1 -18303.651,E2 -18303.651} C_VEL
LIN {X 0,Y 263.137,Z 258.07,A -85,B 0,C 180,E1 -18307.898,E2 -18307.898} C_VEL
LIN {X 0,Y 263.158,Z 256.808,A -85,B 0,C 180,E1 -18309.86,E2 -18309.86} C_VEL
LIN {X 0,Y 263.061,Z 255.717,A -85,B 0,C 180,E1 -18311.902,E2 -18311.902} C_VEL
LIN {X 0,Y 263.098,Z 255.714,A -85,B 0,C 180,E1 -18316.153,E2 -18316.153} C_VEL
LIN {X 0,Y 263.108,Z 255.712,A -85,B 0,C 180,E1 -18320.127,E2 -18320.127} C_VEL
LIN {X 0,Y 263.18,Z 255.7,A -85,B 0,C 180,E1 -18324.02,E2 -18324.02} C_VEL
LIN {X 0,Y 263.125,Z 255.71,A -85,B 0,C 180,E1 -18327.71,E2 -18327.71} C_VEL
LIN {X 0,Y 263.191,Z 255.699,A -85,B 0,C 180,E1 -18331.782,E2 -18331.782} C_VEL
LIN {X 0,Y 263.216,Z 255.698,A -85,B 0,C 180,E1 -18335.199,E2 -18335.199} C_VEL
LIN {X 0,Y 263.254,Z 255.692,A -85,B 0,C 180,E1 -18339.692,E2 -18339.692} C_VEL
LIN {X 0,Y 263.34,Z 255.683,A -85,B 0,C 180,E1 -18344.521,E2 -18344.521} C_VEL
LIN {X 0,Y 263.363,Z 255.681,A -85,B 0,C 180,E1 -18349.234,E2 -18349.234} C_VEL
LIN {X 0,Y 263.564,Z 255.656,A -85,B 0,C 180,E1 -18352.338,E2 -18352.338} C_VEL
LIN {X 0,Y 263.745,Z 255.632,A -85,B 0,C 180,E1 -18358.473,E2 -18358.473} C_VEL
LIN {X 0,Y 263.74,Z 255.634,A -85,B 0,C 180,E1 -18361.527,E2 -18361.527} C_VEL
LIN {X 0,Y 263.564,Z 255.655,A -85,B 0,C 180,E1 -18367.662,E2 -18367.662} C_VEL
LIN {X 0,Y 263.363,Z 255.678,A -85,B 0,C 180,E1 -18370.766,E2 -18370.766} C_VEL
LIN {X 0,Y 263.34,Z 255.675,A -85,B 0,C 180,E1 -18375.479,E2 -18375.479} C_VEL
LIN {X 0,Y 263.253,Z 255.693,A -85,B 0,C 180,E1 -18380.307,E2 -18380.307} C_VEL
LIN {X 0,Y 263.14,Z 255.706,A -85,B 0,C 180,E1 -18383.041,E2 -18383.041} C_VEL
LIN {X 0,Y 262.521,Z 255.787,A -85,B 0,C 180,E1 -18384.319,E2 -18384.319} C_VEL
LIN {X 0,Y 259.712,Z 256.142,A -85,B 0,C 180,E1 -18386.401,E2 -18386.401} C_VEL
LIN {X 0,Y 257.277,Z 256.444,A -85,B 0,C 180,E1 -18388.094,E2 -18388.094} C_VEL
LIN {X 0,Y 256.193,Z 256.573,A -85,B 0,C 180,E1 -18389.407,E2 -18389.407} C_VEL
LIN {X 0,Y 256.086,Z 256.584,A -85,B 0,C 180,E1 -18389.852,E2 -18389.852} C_VEL
LIN {X 0,Y 256.133,Z 256.742,A -85,B 0,C 180,E1 -18392.632,E2 -18392.632} C_VEL
LIN {X 0,Y 256.799,Z 260.385,A -85,B 0,C 180,E1 -18397.02,E2 -18397.02} C_VEL
LIN {X 0,Y 257.392,Z 264.04,A -85,B 0,C 180,E1 -18400.943,E2 -18400.943} C_VEL
LIN {X 0,Y 258.183,Z 268.151,A -85,B 0,C 180,E1 -18405.052,E2 -18405.052} C_VEL
LIN {X 0,Y 259.061,Z 272.939,A -85,B 0,C 180,E1 -18409.429,E2 -18409.429} C_VEL
LIN {X 0,Y 259.39,Z 275.693,A -85,B 0,C 180,E1 -18411.789,E2 -18411.789} C_VEL
LIN {X 0,Y 259.331,Z 277.69,A -85,B 0,C 180,E1 -18413.404,E2 -18413.404} C_VEL
LIN {X 0,Y 258.011,Z 283.191,A -85,B 0,C 180,E1 -18417.609,E2 -18417.609} C_VEL
LIN {X 0,Y 257.376,Z 286.262,A -85,B 0,C 180,E1 -18419.917,E2 -18419.917} C_VEL
LIN {X 0,Y 258.161,Z 289.532,A -85,B 0,C 180,E1 -18420.174,E2 -18420.174} C_VEL
LIN {X 0,Y 261.422,Z 302.324,A -85,B 0,C 180,E1 -18421.364,E2 -18421.364} C_VEL
LIN {X 0,Y 263.673,Z 314.866,A -85,B 0,C 180,E1 -18422.708,E2 -18422.708} C_VEL
LIN {X 0,Y 264.813,Z 325.502,A -85,B 0,C 180,E1 -18424.02,E2 -18424.02} C_VEL
LIN {X 0,Y 265.178,Z 336.26,A -85,B 0,C 180,E1 -18425.539,E2 -18425.539} C_VEL
LIN {X 0,Y 264.886,Z 343.809,A -85,B 0,C 180,E1 -18426.757,E2 -18426.757} C_VEL
LIN {X 0,Y 262.746,Z 353.345,A -85,B 0,C 180,E1 -18428.423,E2 -18428.423} C_VEL
LIN {X 0,Y 260.703,Z 362.067,A -85,B 0,C 180,E1 -18430.31,E2 -18430.31} C_VEL
LIN {X 0,Y 258.749,Z 370.569,A -85,B 0,C 180,E1 -18432.618,E2 -18432.618} C_VEL
LIN {X 0,Y 257.064,Z 377.417,A -85,B 0,C 180,E1 -18434.949,E2 -18434.949} C_VEL
LIN {X 0,Y 255.703,Z 382.913,A -85,B 0,C 180,E1 -18437.3,E2 -18437.3} C_VEL
LIN {X 0,Y 254.868,Z 387.24,A -85,B 0,C 180,E1 -18439.677,E2 -18439.677} C_VEL
LIN {X 0,Y 254.377,Z 390.51,A -85,B 0,C 180,E1 -18442.062,E2 -18442.062} C_VEL
LIN {X 0,Y 254.167,Z 392.864,A -85,B 0,C 180,E1 -18444.528,E2 -18444.528} C_VEL
LIN {X 0,Y 254.17,Z 394.178,A -85,B 0,C 180,E1 -18446.832,E2 -18446.832} C_VEL
LIN {X 0,Y 254.174,Z 394.567,A -85,B 0,C 180,E1 -18448.418,E2 -18448.418} C_VEL
LIN {X 0,Y 254.259,Z 394.569,A -85,B 0,C 180,E1 -18450.002,E2 -18450.002} C_VEL
LIN {X 0,Y 254.2,Z 394.168,A -85,B 0,C 180,E1 -18451.587,E2 -18451.587} C_VEL
LIN {X 0,Y 254.213,Z 393.334,A -85,B 0,C 180,E1 -18453.172,E2 -18453.172} C_VEL
LIN {X 0,Y 254.2,Z 391.319,A -85,B 0,C 180,E1 -18455.549,E2 -18455.549} C_VEL
LIN {X 0,Y 254.4,Z 388.301,A -85,B 0,C 180,E1 -18457.942,E2 -18457.942} C_VEL
LIN {X 0,Y 254.895,Z 384.231,A -85,B 0,C 180,E1 -18460.327,E2 -18460.327} C_VEL
LIN {X 0,Y 255.863,Z 377.971,A -85,B 0,C 180,E1 -18463.1,E2 -18463.1} C_VEL
LIN {X 0,Y 257.166,Z 371.161,A -85,B 0,C 180,E1 -18465.456,E2 -18465.456} C_VEL
LIN {X 0,Y 258.683,Z 363.142,A -85,B 0,C 180,E1 -18467.683,E2 -18467.683} C_VEL
LIN {X 0,Y 260.345,Z 353.984,A -85,B 0,C 180,E1 -18469.723,E2 -18469.723} C_VEL
LIN {X 0,Y 262.363,Z 343.264,A -85,B 0,C 180,E1 -18471.615,E2 -18471.615} C_VEL
LIN {X 0,Y 262.764,Z 339.497,A -85,B 0,C 180,E1 -18472.199,E2 -18472.199} C_VEL
LIN {X 0,Y 262.329,Z 327.826,A -85,B 0,C 180,E1 -18473.874,E2 -18473.874} C_VEL
LIN {X 0,Y 261.508,Z 315.755,A -85,B 0,C 180,E1 -18475.279,E2 -18475.279} C_VEL
LIN {X 0,Y 259.712,Z 302.384,A -85,B 0,C 180,E1 -18476.544,E2 -18476.544} C_VEL
LIN {X 0,Y 257.006,Z 289.327,A -85,B 0,C 180,E1 -18477.551,E2 -18477.551} C_VEL
LIN {X 0,Y 256.514,Z 286.739,A -85,B 0,C 180,E1 -18477.706,E2 -18477.706} C_VEL
LIN {X 0,Y 257.719,Z 280.465,A -85,B 0,C 180,E1 -18482.288,E2 -18482.288} C_VEL
LIN {X 0,Y 258.6,Z 276.245,A -85,B 0,C 180,E1 -18485.382,E2 -18485.382} C_VEL
LIN {X 0,Y 258.898,Z 272.743,A -85,B 0,C 180,E1 -18488.073,E2 -18488.073} C_VEL
LIN {X 0,Y 258.296,Z 268.419,A -85,B 0,C 180,E1 -18491.685,E2 -18491.685} C_VEL
LIN {X 0,Y 257.488,Z 264.408,A -85,B 0,C 180,E1 -18495.21,E2 -18495.21} C_VEL
LIN {X 0,Y 256.824,Z 260.443,A -85,B 0,C 180,E1 -18498.947,E2 -18498.947} C_VEL
LIN {X 0,Y 256.157,Z 256.578,A -85,B 0,C 180,E1 -18502.872,E2 -18502.872} C_VEL
LIN {X 0,Y 256.073,Z 256.588,A -85,B 0,C 180,E1 -18506.708,E2 -18506.708} C_VEL
LIN {X 0,Y 256.063,Z 256.589,A -85,B 0,C 180,E1 -18510.394,E2 -18510.394} C_VEL
LIN {X 0,Y 256.169,Z 256.574,A -85,B 0,C 180,E1 -18514.876,E2 -18514.876} C_VEL
LIN {X 0,Y 256.156,Z 256.576,A -85,B 0,C 180,E1 -18519.104,E2 -18519.104} C_VEL
LIN {X 0,Y 256.229,Z 256.57,A -85,B 0,C 180,E1 -18524.081,E2 -18524.081} C_VEL
LIN {X 0,Y 256.282,Z 256.561,A -85,B 0,C 180,E1 -18528.933,E2 -18528.933} C_VEL
LIN {X 0,Y 256.513,Z 256.531,A -85,B 0,C 180,E1 -18532.126,E2 -18532.126} C_VEL
LIN {X 0,Y 256.504,Z 256.53,A -85,B 0,C 180,E1 -18536.859,E2 -18536.859} C_VEL
LIN {X 0,Y 256.758,Z 256.498,A -85,B 0,C 180,E1 -18540,E2 -18540} C_VEL
LIN {X 0,Y 256.465,Z 256.539,A -85,B 0,C 180,E1 -18543.142,E2 -18543.142} C_VEL
LIN {X 0,Y 256.476,Z 256.536,A -85,B 0,C 180,E1 -18547.875,E2 -18547.875} C_VEL
LIN {X 0,Y 256.299,Z 256.558,A -85,B 0,C 180,E1 -18551.067,E2 -18551.067} C_VEL
LIN {X 0,Y 256.254,Z 256.562,A -85,B 0,C 180,E1 -18555.918,E2 -18555.918} C_VEL
LIN {X 0,Y 256.153,Z 256.577,A -85,B 0,C 180,E1 -18560.897,E2 -18560.897} C_VEL
LIN {X 0,Y 256.091,Z 256.585,A -85,B 0,C 180,E1 -18565.087,E2 -18565.087} C_VEL
LIN {X 0,Y 256.085,Z 256.585,A -85,B 0,C 180,E1 -18568.569,E2 -18568.569} C_VEL
LIN {X 0,Y 256.078,Z 256.585,A -85,B 0,C 180,E1 -18571.699,E2 -18571.699} C_VEL
LIN {X 0,Y 256.091,Z 256.584,A -85,B 0,C 180,E1 -18575.192,E2 -18575.192} C_VEL
LIN {X 0,Y 256.123,Z 256.579,A -85,B 0,C 180,E1 -18577.27,E2 -18577.27} C_VEL
LIN {X 0,Y 256.063,Z 256.587,A -85,B 0,C 180,E1 -18581.202,E2 -18581.202} C_VEL
LIN {X 0,Y 256.045,Z 256.589,A -85,B 0,C 180,E1 -18585.534,E2 -18585.534} C_VEL
LIN {X 0,Y 256.016,Z 256.594,A -85,B 0,C 180,E1 -18588.786,E2 -18588.786} C_VEL
LIN {X 0,Y 256.105,Z 256.582,A -85,B 0,C 180,E1 -18592.861,E2 -18592.861} C_VEL
LIN {X 0,Y 256.013,Z 256.592,A -85,B 0,C 180,E1 -18596.697,E2 -18596.697} C_VEL
LIN {X 0,Y 255.742,Z 256.624,A -85,B 0,C 180,E1 -18600.351,E2 -18600.351} C_VEL
LIN {X 0,Y 255.701,Z 257.576,A -85,B 0,C 180,E1 -18602.142,E2 -18602.142} C_VEL
LIN {X 0,Y 255.488,Z 260.827,A -85,B 0,C 180,E1 -18606.584,E2 -18606.584} C_VEL
LIN {X 0,Y 260.178,Z 274.702,A -85,B 0,C 180,E1 -18607.894,E2 -18607.894} C_VEL
LIN {X 0,Y 263.213,Z 286.071,A -85,B 0,C 180,E1 -18609.153,E2 -18609.153} C_VEL
LIN {X 0,Y 265.402,Z 297.353,A -85,B 0,C 180,E1 -18610.597,E2 -18610.597} C_VEL
LIN {X 0,Y 265.776,Z 299.992,A -85,B 0,C 180,E1 -18610.975,E2 -18610.975} C_VEL
LIN {X 0,Y 264.22,Z 310.613,A -85,B 0,C 180,E1 -18612.386,E2 -18612.386} C_VEL
LIN {X 0,Y 262.598,Z 320.734,A -85,B 0,C 180,E1 -18614.076,E2 -18614.076} C_VEL
LIN {X 0,Y 260.818,Z 329.845,A -85,B 0,C 180,E1 -18615.963,E2 -18615.963} C_VEL
LIN {X 0,Y 259.395,Z 337.349,A -85,B 0,C 180,E1 -18617.877,E2 -18617.877} C_VEL
LIN {X 0,Y 257.827,Z 344.719,A -85,B 0,C 180,E1 -18620.189,E2 -18620.189} C_VEL
LIN {X 0,Y 256.846,Z 349.736,A -85,B 0,C 180,E1 -18622.134,E2 -18622.134} C_VEL
LIN {X 0,Y 255.828,Z 354.609,A -85,B 0,C 180,E1 -18624.48,E2 -18624.48} C_VEL
LIN {X 0,Y 255.094,Z 358.377,A -85,B 0,C 180,E1 -18626.839,E2 -18626.839} C_VEL
LIN {X 0,Y 254.78,Z 360.318,A -85,B 0,C 180,E1 -18628.417,E2 -18628.417} C_VEL
LIN {X 0,Y 254.551,Z 361.856,A -85,B 0,C 180,E1 -18629.998,E2 -18629.998} C_VEL
LIN {X 0,Y 254.408,Z 362.964,A -85,B 0,C 180,E1 -18631.581,E2 -18631.581} C_VEL
LIN {X 0,Y 254.48,Z 363.983,A -85,B 0,C 180,E1 -18634.75,E2 -18634.75} C_VEL
LIN {X 0,Y 254.605,Z 363.923,A -85,B 0,C 180,E1 -18636.417,E2 -18636.417} C_VEL
LIN {X 0,Y 254.926,Z 362.608,A -85,B 0,C 180,E1 -18639.519,E2 -18639.519} C_VEL
LIN {X 0,Y 255.762,Z 359.689,A -85,B 0,C 180,E1 -18642.697,E2 -18642.697} C_VEL
LIN {X 0,Y 256.814,Z 356.327,A -85,B 0,C 180,E1 -18645.066,E2 -18645.066} C_VEL
LIN {X 0,Y 258.319,Z 351.104,A -85,B 0,C 180,E1 -18647.779,E2 -18647.779} C_VEL
LIN {X 0,Y 260.027,Z 345.108,A -85,B 0,C 180,E1 -18650.155,E2 -18650.155} C_VEL
LIN {X 0,Y 262.074,Z 337.726,A -85,B 0,C 180,E1 -18652.464,E2 -18652.464} C_VEL
LIN {X 0,Y 263.998,Z 330.173,A -85,B 0,C 180,E1 -18654.368,E2 -18654.368} C_VEL
LIN {X 0,Y 265.848,Z 321.906,A -85,B 0,C 180,E1 -18656.085,E2 -18656.085} C_VEL
LIN {X 0,Y 268.031,Z 312.017,A -85,B 0,C 180,E1 -18657.735,E2 -18657.735} C_VEL
LIN {X 0,Y 269.213,Z 305.195,A -85,B 0,C 180,E1 -18658.687,E2 -18658.687} C_VEL
LIN {X 0,Y 267.539,Z 295.803,A -85,B 0,C 180,E1 -18660.163,E2 -18660.163} C_VEL
LIN {X 0,Y 265.083,Z 285.938,A -85,B 0,C 180,E1 -18661.564,E2 -18661.564} C_VEL
LIN {X 0,Y 261.12,Z 274.089,A -85,B 0,C 180,E1 -18663.098,E2 -18663.098} C_VEL
LIN {X 0,Y 257.065,Z 264.437,A -85,B 0,C 180,E1 -18664.255,E2 -18664.255} C_VEL
LIN {X 0,Y 256.02,Z 261.437,A -85,B 0,C 180,E1 -18664.597,E2 -18664.597} C_VEL
LIN {X 0,Y 256.134,Z 259.653,A -85,B 0,C 180,E1 -18667.276,E2 -18667.276} C_VEL
LIN {X 0,Y 256.176,Z 258.032,A -85,B 0,C 180,E1 -18669.81,E2 -18669.81} C_VEL
LIN {X 0,Y 256.018,Z 256.629,A -85,B 0,C 180,E1 -18672.167,E2 -18672.167} C_VEL
LIN {X 0,Y 256.042,Z 256.593,A -85,B 0,C 180,E1 -18676.668,E2 -18676.668} C_VEL
LIN {X 0,Y 256.081,Z 256.586,A -85,B 0,C 180,E1 -18680.859,E2 -18680.859} C_VEL
LIN {X 0,Y 256.113,Z 256.583,A -85,B 0,C 180,E1 -18684.811,E2 -18684.811} C_VEL
LIN {X 0,Y 256.083,Z 256.584,A -85,B 0,C 180,E1 -18688.571,E2 -18688.571} C_VEL
LIN {X 0,Y 256.132,Z 256.575,A -85,B 0,C 180,E1 -18692.195,E2 -18692.195} C_VEL
LIN {X 0,Y 256.158,Z 256.577,A -85,B 0,C 180,E1 -18695.698,E2 -18695.698} C_VEL
LIN {X 0,Y 256.157,Z 256.577,A -85,B 0,C 180,E1 -18699.104,E2 -18699.104} C_VEL
LIN {X 0,Y 256.29,Z 256.56,A -85,B 0,C 180,E1 -18704.084,E2 -18704.084} C_VEL
LIN {X 0,Y 256.299,Z 256.559,A -85,B 0,C 180,E1 -18708.933,E2 -18708.933} C_VEL
LIN {X 0,Y 256.531,Z 256.533,A -85,B 0,C 180,E1 -18712.127,E2 -18712.127} C_VEL
LIN {X 0,Y 256.709,Z 256.508,A -85,B 0,C 180,E1 -18718.431,E2 -18718.431} C_VEL
LIN {X 0,Y 256.703,Z 256.51,A -85,B 0,C 180,E1 -18721.569,E2 -18721.569} C_VEL
LIN {X 0,Y 256.531,Z 256.531,A -85,B 0,C 180,E1 -18727.873,E2 -18727.873} C_VEL
LIN {X 0,Y 256.299,Z 256.558,A -85,B 0,C 180,E1 -18731.066,E2 -18731.066} C_VEL
LIN {X 0,Y 256.289,Z 256.553,A -85,B 0,C 180,E1 -18735.916,E2 -18735.916} C_VEL
LIN {X 0,Y 256.156,Z 256.578,A -85,B 0,C 180,E1 -18740.896,E2 -18740.896} C_VEL
LIN {X 0,Y 256.179,Z 256.576,A -85,B 0,C 180,E1 -18745.14,E2 -18745.14} C_VEL
LIN {X 0,Y 256.105,Z 256.584,A -85,B 0,C 180,E1 -18749.601,E2 -18749.601} C_VEL
LIN {X 0,Y 256.086,Z 256.584,A -85,B 0,C 180,E1 -18749.852,E2 -18749.852} C_VEL
LIN {X 0,Y 255.418,Z 256.898,A -85,B 0,C 180,E1 -18751.164,E2 -18751.164} C_VEL
LIN {X 0,Y 252.797,Z 258.413,A -85,B 0,C 180,E1 -18753.292,E2 -18753.292} C_VEL
LIN {X 0,Y 250.654,Z 260.089,A -85,B 0,C 180,E1 -18755.011,E2 -18755.011} C_VEL
LIN {X 0,Y 249.814,Z 261.364,A -85,B 0,C 180,E1 -18756.337,E2 -18756.337} C_VEL
LIN {X 0,Y 249.785,Z 261.76,A -85,B 0,C 180,E1 -18756.785,E2 -18756.785} C_VEL
LIN {X 0,Y 250.416,Z 265.271,A -85,B 0,C 180,E1 -18760.737,E2 -18760.737} C_VEL
LIN {X 0,Y 251.099,Z 268.827,A -85,B 0,C 180,E1 -18764.405,E2 -18764.405} C_VEL
LIN {X 0,Y 251.962,Z 273.542,A -85,B 0,C 180,E1 -18768.861,E2 -18768.861} C_VEL
LIN {X 0,Y 252.338,Z 277.33,A -85,B 0,C 180,E1 -18772.216,E2 -18772.216} C_VEL
LIN {X 0,Y 252.072,Z 279.704,A -85,B 0,C 180,E1 -18774.165,E2 -18774.165} C_VEL
LIN {X 0,Y 250.579,Z 285.716,A -85,B 0,C 180,E1 -18778.874,E2 -18778.874} C_VEL
LIN {X 0,Y 250.61,Z 286.372,A -85,B 0,C 180,E1 -18778.977,E2 -18778.977} C_VEL
LIN {X 0,Y 254.179,Z 299.467,A -85,B 0,C 180,E1 -18780.218,E2 -18780.218} C_VEL
LIN {X 0,Y 256.572,Z 311.825,A -85,B 0,C 180,E1 -18781.566,E2 -18781.566} C_VEL
LIN {X 0,Y 257.922,Z 322.128,A -85,B 0,C 180,E1 -18782.847,E2 -18782.847} C_VEL
LIN {X 0,Y 258.56,Z 333.717,A -85,B 0,C 180,E1 -18784.494,E2 -18784.494} C_VEL
LIN {X 0,Y 258.288,Z 343.689,A -85,B 0,C 180,E1 -18786.127,E2 -18786.127} C_VEL
LIN {X 0,Y 256.14,Z 353.173,A -85,B 0,C 180,E1 -18787.838,E2 -18787.838} C_VEL
LIN {X 0,Y 253.981,Z 361.85,A -85,B 0,C 180,E1 -18789.766,E2 -18789.766} C_VEL
LIN {X 0,Y 251.965,Z 370.302,A -85,B 0,C 180,E1 -18792.135,E2 -18792.135} C_VEL
LIN {X 0,Y 250.195,Z 377.12,A -85,B 0,C 180,E1 -18794.525,E2 -18794.525} C_VEL
LIN {X 0,Y 248.739,Z 382.589,A -85,B 0,C 180,E1 -18796.939,E2 -18796.939} C_VEL
LIN {X 0,Y 247.848,Z 386.891,A -85,B 0,C 180,E1 -18799.381,E2 -18799.381} C_VEL
LIN {X 0,Y 247.333,Z 390.139,A -85,B 0,C 180,E1 -18801.835,E2 -18801.835} C_VEL
LIN {X 0,Y 247.087,Z 392.618,A -85,B 0,C 180,E1 -18804.575,E2 -18804.575} C_VEL
LIN {X 0,Y 247.081,Z 393.766,A -85,B 0,C 180,E1 -18806.741,E2 -18806.741} C_VEL
LIN {X 0,Y 247.1,Z 394.146,A -85,B 0,C 180,E1 -18808.373,E2 -18808.373} C_VEL
LIN {X 0,Y 247.179,Z 394.137,A -85,B 0,C 180,E1 -18810.002,E2 -18810.002} C_VEL
LIN {X 0,Y 247.126,Z 393.724,A -85,B 0,C 180,E1 -18811.632,E2 -18811.632} C_VEL
LIN {X 0,Y 247.122,Z 392.869,A -85,B 0,C 180,E1 -18813.263,E2 -18813.263} C_VEL
LIN {X 0,Y 247.13,Z 391.021,A -85,B 0,C 180,E1 -18815.53,E2 -18815.53} C_VEL
LIN {X 0,Y 247.356,Z 387.796,A -85,B 0,C 180,E1 -18818.17,E2 -18818.17} C_VEL
LIN {X 0,Y 247.865,Z 383.7,A -85,B 0,C 180,E1 -18820.623,E2 -18820.623} C_VEL
LIN {X 0,Y 248.893,Z 377.407,A -85,B 0,C 180,E1 -18823.474,E2 -18823.474} C_VEL
LIN {X 0,Y 250.24,Z 370.565,A -85,B 0,C 180,E1 -18825.895,E2 -18825.895} C_VEL
LIN {X 0,Y 251.665,Z 363.594,A -85,B 0,C 180,E1 -18827.892,E2 -18827.892} C_VEL
LIN {X 0,Y 253.272,Z 355.192,A -85,B 0,C 180,E1 -18829.875,E2 -18829.875} C_VEL
LIN {X 0,Y 255.264,Z 344.889,A -85,B 0,C 180,E1 -18831.822,E2 -18831.822} C_VEL
LIN {X 0,Y 255.913,Z 340.026,A -85,B 0,C 180,E1 -18832.613,E2 -18832.613} C_VEL
LIN {X 0,Y 255.546,Z 328.316,A -85,B 0,C 180,E1 -18834.366,E2 -18834.366} C_VEL
LIN {X 0,Y 254.875,Z 317.098,A -85,B 0,C 180,E1 -18835.742,E2 -18835.742} C_VEL
LIN {X 0,Y 253.258,Z 304.28,A -85,B 0,C 180,E1 -18837.05,E2 -18837.05} C_VEL
LIN {X 0,Y 250.62,Z 291.113,A -85,B 0,C 180,E1 -18838.146,E2 -18838.146} C_VEL
LIN {X 0,Y 249.639,Z 286.292,A -85,B 0,C 180,E1 -18838.492,E2 -18838.492} C_VEL
LIN {X 0,Y 250.775,Z 280.605,A -85,B 0,C 180,E1 -18842.78,E2 -18842.78} C_VEL
LIN {X 0,Y 251.643,Z 276.476,A -85,B 0,C 180,E1 -18845.911,E2 -18845.911} C_VEL
LIN {X 0,Y 251.846,Z 273.129,A -85,B 0,C 180,E1 -18848.614,E2 -18848.614} C_VEL
LIN {X 0,Y 251.165,Z 268.994,A -85,B 0,C 180,E1 -18852.19,E2 -18852.19} C_VEL
LIN {X 0,Y 250.192,Z 263.89,A -85,B 0,C 180,E1 -18856.919,E2 -18856.919} C_VEL
LIN {X 0,Y 249.713,Z 261.102,A -85,B 0,C 180,E1 -18859.66,E2 -18859.66} C_VEL
LIN {X 0,Y 249.06,Z 257.462,A -85,B 0,C 180,E1 -18863.534,E2 -18863.534} C_VEL
LIN {X 0,Y 249.041,Z 257.463,A -85,B 0,C 180,E1 -18867.849,E2 -18867.849} C_VEL
LIN {X 0,Y 249.057,Z 257.459,A -85,B 0,C 180,E1 -18871.333,E2 -18871.333} C_VEL
LIN {X 0,Y 249.134,Z 257.45,A -85,B 0,C 180,E1 -18874.967,E2 -18874.967} C_VEL
LIN {X 0,Y 249.098,Z 257.457,A -85,B 0,C 180,E1 -18878.606,E2 -18878.606} C_VEL
LIN {X 0,Y 249.166,Z 257.449,A -85,B 0,C 180,E1 -18883.617,E2 -18883.617} C_VEL
LIN {X 0,Y 249.226,Z 257.441,A -85,B 0,C 180,E1 -18888.615,E2 -18888.615} C_VEL
LIN {X 0,Y 249.451,Z 257.412,A -85,B 0,C 180,E1 -18891.902,E2 -18891.902} C_VEL
LIN {X 0,Y 249.3,Z 257.431,A -85,B 0,C 180,E1 -18895.149,E2 -18895.149} C_VEL
LIN {X 0,Y 249.683,Z 257.382,A -85,B 0,C 180,E1 -18898.387,E2 -18898.387} C_VEL
LIN {X 0,Y 249.671,Z 257.386,A -85,B 0,C 180,E1 -18901.613,E2 -18901.613} C_VEL
LIN {X 0,Y 249.428,Z 257.412,A -85,B 0,C 180,E1 -18906.567,E2 -18906.567} C_VEL
LIN {X 0,Y 249.352,Z 257.421,A -85,B 0,C 180,E1 -18909.736,E2 -18909.736} C_VEL
LIN {X 0,Y 249.184,Z 257.443,A -85,B 0,C 180,E1 -18914.705,E2 -18914.705} C_VEL
LIN {X 0,Y 249.117,Z 257.452,A -85,B 0,C 180,E1 -18918.079,E2 -18918.079} C_VEL
LIN {X 0,Y 249.086,Z 257.457,A -85,B 0,C 180,E1 -18921.519,E2 -18921.519} C_VEL
LIN {X 0,Y 249.052,Z 257.46,A -85,B 0,C 180,E1 -18925.439,E2 -18925.439} C_VEL
LIN {X 0,Y 249.033,Z 257.462,A -85,B 0,C 180,E1 -18928.968,E2 -18928.968} C_VEL
LIN {X 0,Y 249.034,Z 257.464,A -85,B 0,C 180,E1 -18932.426,E2 -18932.426} C_VEL
LIN {X 0,Y 249.057,Z 257.462,A -85,B 0,C 180,E1 -18936.341,E2 -18936.341} C_VEL
LIN {X 0,Y 249.014,Z 257.467,A -85,B 0,C 180,E1 -18940.477,E2 -18940.477} C_VEL
LIN {X 0,Y 248.991,Z 257.468,A -85,B 0,C 180,E1 -18944.882,E2 -18944.882} C_VEL
LIN {X 0,Y 248.991,Z 257.469,A -85,B 0,C 180,E1 -18947.355,E2 -18947.355} C_VEL
LIN {X 0,Y 249.027,Z 257.467,A -85,B 0,C 180,E1 -18952.206,E2 -18952.206} C_VEL
LIN {X 0,Y 249.017,Z 257.467,A -85,B 0,C 180,E1 -18955.633,E2 -18955.633} C_VEL
LIN {X 0,Y 248.769,Z 257.492,A -85,B 0,C 180,E1 -18959.432,E2 -18959.432} C_VEL
LIN {X 0,Y 248.67,Z 258.064,A -85,B 0,C 180,E1 -18961.282,E2 -18961.282} C_VEL
LIN {X 0,Y 248.525,Z 261.309,A -85,B 0,C 180,E1 -18965.817,E2 -18965.817} C_VEL
LIN {X 0,Y 251.323,Z 269.413,A -85,B 0,C 180,E1 -18966.574,E2 -18966.574} C_VEL
LIN {X 0,Y 254.886,Z 280.646,A -85,B 0,C 180,E1 -18967.794,E2 -18967.794} C_VEL
LIN {X 0,Y 257.591,Z 292.221,A -85,B 0,C 180,E1 -18969.223,E2 -18969.223} C_VEL
LIN {X 0,Y 259.061,Z 301.003,A -85,B 0,C 180,E1 -18970.468,E2 -18970.468} C_VEL
LIN {X 0,Y 257.522,Z 311.47,A -85,B 0,C 180,E1 -18971.912,E2 -18971.912} C_VEL
LIN {X 0,Y 255.832,Z 321.494,A -85,B 0,C 180,E1 -18973.643,E2 -18973.643} C_VEL
LIN {X 0,Y 253.987,Z 330.542,A -85,B 0,C 180,E1 -18975.577,E2 -18975.577} C_VEL
LIN {X 0,Y 252.511,Z 338.001,A -85,B 0,C 180,E1 -18977.541,E2 -18977.541} C_VEL
LIN {X 0,Y 250.863,Z 345.333,A -85,B 0,C 180,E1 -18979.913,E2 -18979.913} C_VEL
LIN {X 0,Y 249.839,Z 350.314,A -85,B 0,C 180,E1 -18981.912,E2 -18981.912} C_VEL
LIN {X 0,Y 248.807,Z 355.153,A -85,B 0,C 180,E1 -18984.324,E2 -18984.324} C_VEL
LIN {X 0,Y 248.023,Z 358.893,A -85,B 0,C 180,E1 -18986.749,E2 -18986.749} C_VEL
LIN {X 0,Y 247.697,Z 360.82,A -85,B 0,C 180,E1 -18988.372,E2 -18988.372} C_VEL
LIN {X 0,Y 247.461,Z 362.342,A -85,B 0,C 180,E1 -18989.998,E2 -18989.998} C_VEL
LIN {X 0,Y 247.329,Z 364.108,A -85,B 0,C 180,E1 -18993.256,E2 -18993.256} C_VEL
LIN {X 0,Y 247.533,Z 364.361,A -85,B 0,C 180,E1 -18996.417,E2 -18996.417} C_VEL
LIN {X 0,Y 247.642,Z 363.873,A -85,B 0,C 180,E1 -18998.155,E2 -18998.155} C_VEL
LIN {X 0,Y 248.303,Z 361.715,A -85,B 0,C 180,E1 -19001.425,E2 -19001.425} C_VEL
LIN {X 0,Y 249.12,Z 359.002,A -85,B 0,C 180,E1 -19003.872,E2 -19003.872} C_VEL
LIN {X 0,Y 250.344,Z 355.261,A -85,B 0,C 180,E1 -19006.301,E2 -19006.301} C_VEL
LIN {X 0,Y 252.043,Z 349.58,A -85,B 0,C 180,E1 -19009.081,E2 -19009.081} C_VEL
LIN {X 0,Y 254.036,Z 343.064,A -85,B 0,C 180,E1 -19011.501,E2 -19011.501} C_VEL
LIN {X 0,Y 256.242,Z 335.046,A -85,B 0,C 180,E1 -19013.86,E2 -19013.86} C_VEL
LIN {X 0,Y 258.345,Z 326.835,A -85,B 0,C 180,E1 -19015.799,E2 -19015.799} C_VEL
LIN {X 0,Y 260.68,Z 316.762,A -85,B 0,C 180,E1 -19017.712,E2 -19017.712} C_VEL
LIN {X 0,Y 262.622,Z 307.685,A -85,B 0,C 180,E1 -19019.084,E2 -19019.084} C_VEL
LIN {X 0,Y 261.653,Z 300.421,A -85,B 0,C 180,E1 -19020.283,E2 -19020.283} C_VEL
LIN {X 0,Y 259.452,Z 290.356,A -85,B 0,C 180,E1 -19021.829,E2 -19021.829} C_VEL
LIN {X 0,Y 255.884,Z 278.928,A -85,B 0,C 180,E1 -19023.445,E2 -19023.445} C_VEL
LIN {X 0,Y 251.538,Z 268.074,A -85,B 0,C 180,E1 -19024.864,E2 -19024.864} C_VEL
LIN {X 0,Y 249.096,Z 262.386,A -85,B 0,C 180,E1 -19025.541,E2 -19025.541} C_VEL
LIN {X 0,Y 249.037,Z 261.912,A -85,B 0,C 180,E1 -19025.611,E2 -19025.611} C_VEL
LIN {X 0,Y 249.123,Z 260.17,A -85,B 0,C 180,E1 -19028.36,E2 -19028.36} C_VEL
LIN {X 0,Y 249.114,Z 258.876,A -85,B 0,C 180,E1 -19030.453,E2 -19030.453} C_VEL
LIN {X 0,Y 248.965,Z 257.541,A -85,B 0,C 180,E1 -19032.781,E2 -19032.781} C_VEL
LIN {X 0,Y 249.002,Z 257.468,A -85,B 0,C 180,E1 -19037.359,E2 -19037.359} C_VEL
LIN {X 0,Y 249.031,Z 257.464,A -85,B 0,C 180,E1 -19041.62,E2 -19041.62} C_VEL
LIN {X 0,Y 249.053,Z 257.46,A -85,B 0,C 180,E1 -19045.64,E2 -19045.64} C_VEL
LIN {X 0,Y 249.043,Z 257.459,A -85,B 0,C 180,E1 -19049.472,E2 -19049.472} C_VEL
LIN {X 0,Y 249.064,Z 257.456,A -85,B 0,C 180,E1 -19053.161,E2 -19053.161} C_VEL
LIN {X 0,Y 249.07,Z 257.46,A -85,B 0,C 180,E1 -19056.731,E2 -19056.731} C_VEL
LIN {X 0,Y 249.101,Z 257.456,A -85,B 0,C 180,E1 -19060.21,E2 -19060.21} C_VEL
LIN {X 0,Y 249.232,Z 257.44,A -85,B 0,C 180,E1 -19063.621,E2 -19063.621} C_VEL
LIN {X 0,Y 249.242,Z 257.437,A -85,B 0,C 180,E1 -19068.616,E2 -19068.616} C_VEL
LIN {X 0,Y 249.475,Z 257.41,A -85,B 0,C 180,E1 -19071.902,E2 -19071.902} C_VEL
LIN {X 0,Y 249.452,Z 257.414,A -85,B 0,C 180,E1 -19076.77,E2 -19076.77} C_VEL
LIN {X 0,Y 249.71,Z 257.38,A -85,B 0,C 180,E1 -19080,E2 -19080} C_VEL
LIN {X 0,Y 249.429,Z 257.416,A -85,B 0,C 180,E1 -19083.23,E2 -19083.23} C_VEL
LIN {X 0,Y 249.475,Z 257.41,A -85,B 0,C 180,E1 -19088.097,E2 -19088.097} C_VEL
LIN {X 0,Y 249.242,Z 257.437,A -85,B 0,C 180,E1 -19091.384,E2 -19091.384} C_VEL
LIN {X 0,Y 249.231,Z 257.434,A -85,B 0,C 180,E1 -19096.379,E2 -19096.379} C_VEL
LIN {X 0,Y 249.077,Z 257.459,A -85,B 0,C 180,E1 -19101.519,E2 -19101.519} C_VEL
LIN {X 0,Y 249.121,Z 257.454,A -85,B 0,C 180,E1 -19105.483,E2 -19105.483} C_VEL
LIN {X 0,Y 249.035,Z 257.463,A -85,B 0,C 180,E1 -19109.847,E2 -19109.847} C_VEL
LIN {X 0,Y 249.071,Z 257.571,A -85,B 0,C 180,E1 -19111.577,E2 -19111.577} C_VEL
LIN {X 0,Y 249.61,Z 260.485,A -85,B 0,C 180,E1 -19115.267,E2 -19115.267} C_VEL
LIN {X 0,Y 249.785,Z 261.76,A -85,B 0,C 180,E1 -19116.785,E2 -19116.785} C_VEL
LIN {X 0,Y 249.318,Z 263.038,A -85,B 0,C 180,E1 -19118.103,E2 -19118.103} C_VEL
LIN {X 0,Y 246.922,Z 265.533,A -85,B 0,C 180,E1 -19120.246,E2 -19120.246} C_VEL
LIN {X 0,Y 244.219,Z 268.627,A -85,B 0,C 180,E1 -19122.874,E2 -19122.874} C_VEL
LIN {X 0,Y 244.023,Z 269.567,A -85,B 0,C 180,E1 -19123.781,E2 -19123.781} C_VEL
LIN {X 0,Y 244.851,Z 274.09,A -85,B 0,C 180,E1 -19128.269,E2 -19128.269} C_VEL
LIN {X 0,Y 245.274,Z 276.968,A -85,B 0,C 180,E1 -19130.925,E2 -19130.925} C_VEL
LIN {X 0,Y 245.23,Z 279.761,A -85,B 0,C 180,E1 -19133.364,E2 -19133.364} C_VEL
LIN {X 0,Y 244.104,Z 284.022,A -85,B 0,C 180,E1 -19136.84,E2 -19136.84} C_VEL
LIN {X 0,Y 243.787,Z 285.328,A -85,B 0,C 180,E1 -19137.891,E2 -19137.891} C_VEL
LIN {X 0,Y 244.723,Z 288.947,A -85,B 0,C 180,E1 -19138.226,E2 -19138.226} C_VEL
LIN {X 0,Y 248.145,Z 301.966,A -85,B 0,C 180,E1 -19139.582,E2 -19139.582} C_VEL
LIN {X 0,Y 250.304,Z 313.973,A -85,B 0,C 180,E1 -19140.987,E2 -19140.987} C_VEL
LIN {X 0,Y 251.514,Z 324.46,A -85,B 0,C 180,E1 -19142.39,E2 -19142.39} C_VEL
LIN {X 0,Y 251.975,Z 335.276,A -85,B 0,C 180,E1 -19144.029,E2 -19144.029} C_VEL
LIN {X 0,Y 251.391,Z 345.845,A -85,B 0,C 180,E1 -19145.869,E2 -19145.869} C_VEL
LIN {X 0,Y 248.596,Z 356.636,A -85,B 0,C 180,E1 -19148.004,E2 -19148.004} C_VEL
LIN {X 0,Y 246.537,Z 364.628,A -85,B 0,C 180,E1 -19149.999,E2 -19149.999} C_VEL
LIN {X 0,Y 244.475,Z 372.483,A -85,B 0,C 180,E1 -19152.434,E2 -19152.434} C_VEL
LIN {X 0,Y 242.764,Z 378.785,A -85,B 0,C 180,E1 -19154.9,E2 -19154.9} C_VEL
LIN {X 0,Y 241.445,Z 383.819,A -85,B 0,C 180,E1 -19157.393,E2 -19157.393} C_VEL
LIN {X 0,Y 240.619,Z 387.738,A -85,B 0,C 180,E1 -19159.909,E2 -19159.909} C_VEL
LIN {X 0,Y 240.08,Z 391.387,A -85,B 0,C 180,E1 -19163.278,E2 -19163.278} C_VEL
LIN {X 0,Y 239.988,Z 392.59,A -85,B 0,C 180,E1 -19164.962,E2 -19164.962} C_VEL
LIN {X 0,Y 239.994,Z 393.353,A -85,B 0,C 180,E1 -19166.645,E2 -19166.645} C_VEL
LIN {X 0,Y 240.027,Z 393.725,A -85,B 0,C 180,E1 -19168.325,E2 -19168.325} C_VEL
LIN {X 0,Y 240.101,Z 393.705,A -85,B 0,C 180,E1 -19170.002,E2 -19170.002} C_VEL
LIN {X 0,Y 240.052,Z 393.278,A -85,B 0,C 180,E1 -19171.68,E2 -19171.68} C_VEL
LIN {X 0,Y 240.033,Z 392.405,A -85,B 0,C 180,E1 -19173.36,E2 -19173.36} C_VEL
LIN {X 0,Y 240.03,Z 390.777,A -85,B 0,C 180,E1 -19175.432,E2 -19175.432} C_VEL
LIN {X 0,Y 240.308,Z 387.288,A -85,B 0,C 180,E1 -19178.411,E2 -19178.411} C_VEL
LIN {X 0,Y 240.854,Z 383.167,A -85,B 0,C 180,E1 -19180.936,E2 -19180.936} C_VEL
LIN {X 0,Y 241.957,Z 376.845,A -85,B 0,C 180,E1 -19183.867,E2 -19183.867} C_VEL
LIN {X 0,Y 243.357,Z 369.97,A -85,B 0,C 180,E1 -19186.357,E2 -19186.357} C_VEL
LIN {X 0,Y 244.812,Z 362.961,A -85,B 0,C 180,E1 -19188.411,E2 -19188.411} C_VEL
LIN {X 0,Y 246.544,Z 354.523,A -85,B 0,C 180,E1 -19190.441,E2 -19190.441} C_VEL
LIN {X 0,Y 248.421,Z 345.318,A -85,B 0,C 180,E1 -19192.236,E2 -19192.236} C_VEL
LIN {X 0,Y 249.071,Z 340.546,A -85,B 0,C 180,E1 -19193.051,E2 -19193.051} C_VEL
LIN {X 0,Y 248.81,Z 329.037,A -85,B 0,C 180,E1 -19194.851,E2 -19194.851} C_VEL
LIN {X 0,Y 248.246,Z 318.57,A -85,B 0,C 180,E1 -19196.209,E2 -19196.209} C_VEL
LIN {X 0,Y 246.697,Z 305.471,A -85,B 0,C 180,E1 -19197.636,E2 -19197.636} C_VEL
LIN {X 0,Y 244.234,Z 292.621,A -85,B 0,C 180,E1 -19198.789,E2 -19198.789} C_VEL
LIN {X 0,Y 242.772,Z 285.828,A -85,B 0,C 180,E1 -19199.308,E2 -19199.308} C_VEL
LIN {X 0,Y 244.134,Z 279.668,A -85,B 0,C 180,E1 -19204.151,E2 -19204.151} C_VEL
LIN {X 0,Y 244.798,Z 275.999,A -85,B 0,C 180,E1 -19207.08,E2 -19207.08} C_VEL
LIN {X 0,Y 244.725,Z 273.485,A -85,B 0,C 180,E1 -19209.185,E2 -19209.185} C_VEL
LIN {X 0,Y 244.041,Z 269.54,A -85,B 0,C 180,E1 -19212.748,E2 -19212.748} C_VEL
LIN {X 0,Y 243.154,Z 264.839,A -85,B 0,C 180,E1 -19217.272,E2 -19217.272} C_VEL
LIN {X 0,Y 242.348,Z 259.856,A -85,B 0,C 180,E1 -19222.483,E2 -19222.483} C_VEL
LIN {X 0,Y 241.999,Z 258.342,A -85,B 0,C 180,E1 -19224.491,E2 -19224.491} C_VEL
LIN {X 0,Y 241.961,Z 258.346,A -85,B 0,C 180,E1 -19228.478,E2 -19228.478} C_VEL
LIN {X 0,Y 241.977,Z 258.344,A -85,B 0,C 180,E1 -19232.309,E2 -19232.309} C_VEL
LIN {X 0,Y 242.044,Z 258.335,A -85,B 0,C 180,E1 -19236.015,E2 -19236.015} C_VEL
LIN {X 0,Y 242.024,Z 258.337,A -85,B 0,C 180,E1 -19239.607,E2 -19239.607} C_VEL
LIN {X 0,Y 242.122,Z 258.325,A -85,B 0,C 180,E1 -19243.319,E2 -19243.319} C_VEL
LIN {X 0,Y 242.161,Z 258.322,A -85,B 0,C 180,E1 -19248.279,E2 -19248.279} C_VEL
LIN {X 0,Y 242.398,Z 258.292,A -85,B 0,C 180,E1 -19251.665,E2 -19251.665} C_VEL
LIN {X 0,Y 242.26,Z 258.308,A -85,B 0,C 180,E1 -19255.007,E2 -19255.007} C_VEL
LIN {X 0,Y 242.644,Z 258.259,A -85,B 0,C 180,E1 -19258.34,E2 -19258.34} C_VEL
LIN {X 0,Y 242.631,Z 258.263,A -85,B 0,C 180,E1 -19261.66,E2 -19261.66} C_VEL
LIN {X 0,Y 242.405,Z 258.288,A -85,B 0,C 180,E1 -19266.66,E2 -19266.66} C_VEL
LIN {X 0,Y 242.275,Z 258.302,A -85,B 0,C 180,E1 -19270.024,E2 -19270.024} C_VEL
LIN {X 0,Y 242.143,Z 258.32,A -85,B 0,C 180,E1 -19275.143,E2 -19275.143} C_VEL
LIN {X 0,Y 242.055,Z 258.334,A -85,B 0,C 180,E1 -19278.626,E2 -19278.626} C_VEL
LIN {X 0,Y 241.997,Z 258.34,A -85,B 0,C 180,E1 -19282.182,E2 -19282.182} C_VEL
LIN {X 0,Y 241.995,Z 258.339,A -85,B 0,C 180,E1 -19285.826,E2 -19285.826} C_VEL
LIN {X 0,Y 241.971,Z 258.34,A -85,B 0,C 180,E1 -19289.588,E2 -19289.588} C_VEL
LIN {X 0,Y 241.987,Z 258.338,A -85,B 0,C 180,E1 -19293.492,E2 -19293.492} C_VEL
LIN {X 0,Y 241.998,Z 258.338,A -85,B 0,C 180,E1 -19297.581,E2 -19297.581} C_VEL
LIN {X 0,Y 241.942,Z 258.348,A -85,B 0,C 180,E1 -19301.922,E2 -19301.922} C_VEL
LIN {X 0,Y 241.916,Z 258.351,A -85,B 0,C 180,E1 -19306.576,E2 -19306.576} C_VEL
LIN {X 0,Y 241.981,Z 258.344,A -85,B 0,C 180,E1 -19311.645,E2 -19311.645} C_VEL
LIN {X 0,Y 241.98,Z 258.343,A -85,B 0,C 180,E1 -19314.485,E2 -19314.485} C_VEL
LIN {X 0,Y 241.79,Z 258.361,A -85,B 0,C 180,E1 -19318.45,E2 -19318.45} C_VEL
LIN {X 0,Y 241.649,Z 258.812,A -85,B 0,C 180,E1 -19320.752,E2 -19320.752} C_VEL
LIN {X 0,Y 241.498,Z 261.666,A -85,B 0,C 180,E1 -19324.951,E2 -19324.951} C_VEL
LIN {X 0,Y 246.672,Z 276.513,A -85,B 0,C 180,E1 -19326.525,E2 -19326.525} C_VEL
LIN {X 0,Y 249.747,Z 287.658,A -85,B 0,C 180,E1 -19327.889,E2 -19327.889} C_VEL
LIN {X 0,Y 251.778,Z 298.203,A -85,B 0,C 180,E1 -19329.346,E2 -19329.346} C_VEL
LIN {X 0,Y 252.311,Z 303.32,A -85,B 0,C 180,E1 -19330.112,E2 -19330.112} C_VEL
LIN {X 0,Y 250.679,Z 313.517,A -85,B 0,C 180,E1 -19331.612,E2 -19331.612} C_VEL
LIN {X 0,Y 248.673,Z 324.18,A -85,B 0,C 180,E1 -19333.581,E2 -19333.581} C_VEL
LIN {X 0,Y 247.115,Z 331.496,A -85,B 0,C 180,E1 -19335.234,E2 -19335.234} C_VEL
LIN {X 0,Y 245.34,Z 339.991,A -85,B 0,C 180,E1 -19337.591,E2 -19337.591} C_VEL
LIN {X 0,Y 243.623,Z 347.041,A -85,B 0,C 180,E1 -19340.03,E2 -19340.03} C_VEL
LIN {X 0,Y 242.835,Z 350.892,A -85,B 0,C 180,E1 -19341.677,E2 -19341.677} C_VEL
LIN {X 0,Y 241.788,Z 355.698,A -85,B 0,C 180,E1 -19344.159,E2 -19344.159} C_VEL
LIN {X 0,Y 240.952,Z 359.409,A -85,B 0,C 180,E1 -19346.653,E2 -19346.653} C_VEL
LIN {X 0,Y 240.615,Z 361.322,A -85,B 0,C 180,E1 -19348.324,E2 -19348.324} C_VEL
LIN {X 0,Y 240.372,Z 362.825,A -85,B 0,C 180,E1 -19349.998,E2 -19349.998} C_VEL
LIN {X 0,Y 240.263,Z 364.554,A -85,B 0,C 180,E1 -19353.351,E2 -19353.351} C_VEL
LIN {X 0,Y 240.436,Z 364.803,A -85,B 0,C 180,E1 -19356.364,E2 -19356.364} C_VEL
LIN {X 0,Y 240.603,Z 364.267,A -85,B 0,C 180,E1 -19358.396,E2 -19358.396} C_VEL
LIN {X 0,Y 241.314,Z 362.083,A -85,B 0,C 180,E1 -19361.761,E2 -19361.761} C_VEL
LIN {X 0,Y 242.215,Z 359.34,A -85,B 0,C 180,E1 -19364.276,E2 -19364.276} C_VEL
LIN {X 0,Y 243.482,Z 355.571,A -85,B 0,C 180,E1 -19366.774,E2 -19366.774} C_VEL
LIN {X 0,Y 245.304,Z 349.846,A -85,B 0,C 180,E1 -19369.626,E2 -19369.626} C_VEL
LIN {X 0,Y 247.39,Z 343.285,A -85,B 0,C 180,E1 -19372.109,E2 -19372.109} C_VEL
LIN {X 0,Y 249.734,Z 335.223,A -85,B 0,C 180,E1 -19374.522,E2 -19374.522} C_VEL
LIN {X 0,Y 252.123,Z 326.093,A -85,B 0,C 180,E1 -19376.701,E2 -19376.701} C_VEL
LIN {X 0,Y 254.666,Z 315.62,A -85,B 0,C 180,E1 -19378.65,E2 -19378.65} C_VEL
LIN {X 0,Y 256.046,Z 309.418,A -85,B 0,C 180,E1 -19379.605,E2 -19379.605} C_VEL
LIN {X 0,Y 255.928,Z 306.38,A -85,B 0,C 180,E1 -19380.12,E2 -19380.12} C_VEL
LIN {X 0,Y 253.715,Z 294.741,A -85,B 0,C 180,E1 -19382.084,E2 -19382.084} C_VEL
LIN {X 0,Y 250.523,Z 283.606,A -85,B 0,C 180,E1 -19383.791,E2 -19383.791} C_VEL
LIN {X 0,Y 246.309,Z 272.26,A -85,B 0,C 180,E1 -19385.385,E2 -19385.385} C_VEL
LIN {X 0,Y 242.217,Z 263.23,A -85,B 0,C 180,E1 -19386.593,E2 -19386.593} C_VEL
LIN {X 0,Y 242.06,Z 262.409,A -85,B 0,C 180,E1 -19386.674,E2 -19386.674} C_VEL
LIN {X 0,Y 242.092,Z 260.582,A -85,B 0,C 180,E1 -19389.689,E2 -19389.689} C_VEL
LIN {X 0,Y 241.898,Z 258.464,A -85,B 0,C 180,E1 -19393.419,E2 -19393.419} C_VEL
LIN {X 0,Y 241.932,Z 258.351,A -85,B 0,C 180,E1 -19398.076,E2 -19398.076} C_VEL
LIN {X 0,Y 241.995,Z 258.343,A -85,B 0,C 180,E1 -19402.419,E2 -19402.419} C_VEL
LIN {X 0,Y 241.983,Z 258.34,A -85,B 0,C 180,E1 -19406.507,E2 -19406.507} C_VEL
LIN {X 0,Y 242.028,Z 258.337,A -85,B 0,C 180,E1 -19410.586,E2 -19410.586} C_VEL
LIN {X 0,Y 242.059,Z 258.334,A -85,B 0,C 180,E1 -19414.182,E2 -19414.182} C_VEL
LIN {X 0,Y 242.044,Z 258.335,A -85,B 0,C 180,E1 -19418.296,E2 -19418.296} C_VEL
LIN {X 0,Y 242.153,Z 258.322,A -85,B 0,C 180,E1 -19423.277,E2 -19423.277} C_VEL
LIN {X 0,Y 242.176,Z 258.318,A -85,B 0,C 180,E1 -19428.279,E2 -19428.279} C_VEL
LIN {X 0,Y 242.425,Z 258.288,A -85,B 0,C 180,E1 -19431.665,E2 -19431.665} C_VEL
LIN {X 0,Y 242.255,Z 258.31,A -85,B 0,C 180,E1 -19435.007,E2 -19435.007} C_VEL
LIN {X 0,Y 242.633,Z 258.261,A -85,B 0,C 180,E1 -19438.34,E2 -19438.34} C_VEL
LIN {X 0,Y 242.626,Z 258.264,A -85,B 0,C 180,E1 -19441.66,E2 -19441.66} C_VEL
LIN {X 0,Y 242.425,Z 258.287,A -85,B 0,C 180,E1 -19446.659,E2 -19446.659} C_VEL
LIN {X 0,Y 242.335,Z 258.3,A -85,B 0,C 180,E1 -19450.021,E2 -19450.021} C_VEL
LIN {X 0,Y 242.156,Z 258.314,A -85,B 0,C 180,E1 -19455.141,E2 -19455.141} C_VEL
LIN {X 0,Y 242.063,Z 258.326,A -85,B 0,C 180,E1 -19458.625,E2 -19458.625} C_VEL
LIN {X 0,Y 242.003,Z 258.342,A -85,B 0,C 180,E1 -19462.181,E2 -19462.181} C_VEL
LIN {X 0,Y 242.057,Z 258.333,A -85,B 0,C 180,E1 -19465.839,E2 -19465.839} C_VEL
LIN {X 0,Y 242.041,Z 258.465,A -85,B 0,C 180,E1 -19470.54,E2 -19470.54} C_VEL
LIN {X 0,Y 242.695,Z 262.123,A -85,B 0,C 180,E1 -19475.392,E2 -19475.392} C_VEL
LIN {X 0,Y 243.24,Z 265.592,A -85,B 0,C 180,E1 -19479.468,E2 -19479.468} C_VEL
LIN {X 0,Y 244.023,Z 269.567,A -85,B 0,C 180,E1 -19483.781,E2 -19483.781} C_VEL
LIN {X 0,Y 243.55,Z 271.014,A -85,B 0,C 180,E1 -19485.12,E2 -19485.12} C_VEL
LIN {X 0,Y 241.146,Z 273.707,A -85,B 0,C 180,E1 -19487.3,E2 -19487.3} C_VEL
LIN {X 0,Y 238.422,Z 277.023,A -85,B 0,C 180,E1 -19489.975,E2 -19489.975} C_VEL
LIN {X 0,Y 238.213,Z 278.061,A -85,B 0,C 180,E1 -19490.898,E2 -19490.898} C_VEL
LIN {X 0,Y 238.264,Z 280.149,A -85,B 0,C 180,E1 -19492.789,E2 -19492.789} C_VEL
LIN {X 0,Y 237.151,Z 284.518,A -85,B 0,C 180,E1 -19496.499,E2 -19496.499} C_VEL
LIN {X 0,Y 237.048,Z 284.872,A -85,B 0,C 180,E1 -19496.796,E2 -19496.796} C_VEL
LIN {X 0,Y 237.939,Z 288.337,A -85,B 0,C 180,E1 -19497.122,E2 -19497.122} C_VEL
LIN {X 0,Y 241.503,Z 301.425,A -85,B 0,C 180,E1 -19498.573,E2 -19498.573} C_VEL
LIN {X 0,Y 243.794,Z 314.178,A -85,B 0,C 180,E1 -19500.136,E2 -19500.136} C_VEL
LIN {X 0,Y 244.97,Z 324.808,A -85,B 0,C 180,E1 -19501.625,E2 -19501.625} C_VEL
LIN {X 0,Y 245.366,Z 335.859,A -85,B 0,C 180,E1 -19503.387,E2 -19503.387} C_VEL
LIN {X 0,Y 244.865,Z 345.701,A -85,B 0,C 180,E1 -19505.183,E2 -19505.183} C_VEL
LIN {X 0,Y 242.004,Z 356.445,A -85,B 0,C 180,E1 -19507.372,E2 -19507.372} C_VEL
LIN {X 0,Y 239.852,Z 364.397,A -85,B 0,C 180,E1 -19509.417,E2 -19509.417} C_VEL
LIN {X 0,Y 237.704,Z 372.203,A -85,B 0,C 180,E1 -19511.917,E2 -19511.917} C_VEL
LIN {X 0,Y 235.894,Z 378.476,A -85,B 0,C 180,E1 -19514.449,E2 -19514.449} C_VEL
LIN {X 0,Y 234.464,Z 383.483,A -85,B 0,C 180,E1 -19517.011,E2 -19517.011} C_VEL
LIN {X 0,Y 233.588,Z 387.378,A -85,B 0,C 180,E1 -19519.602,E2 -19519.602} C_VEL
LIN {X 0,Y 233.221,Z 389.397,A -85,B 0,C 180,E1 -19521.337,E2 -19521.337} C_VEL
LIN {X 0,Y 232.912,Z 392.143,A -85,B 0,C 180,E1 -19524.721,E2 -19524.721} C_VEL
LIN {X 0,Y 232.912,Z 392.942,A -85,B 0,C 180,E1 -19526.543,E2 -19526.543} C_VEL
LIN {X 0,Y 232.955,Z 393.303,A -85,B 0,C 180,E1 -19528.274,E2 -19528.274} C_VEL
LIN {X 0,Y 233.025,Z 393.274,A -85,B 0,C 180,E1 -19530.003,E2 -19530.003} C_VEL
LIN {X 0,Y 232.98,Z 392.829,A -85,B 0,C 180,E1 -19531.731,E2 -19531.731} C_VEL
LIN {X 0,Y 232.947,Z 391.94,A -85,B 0,C 180,E1 -19533.462,E2 -19533.462} C_VEL
LIN {X 0,Y 232.954,Z 390.479,A -85,B 0,C 180,E1 -19535.39,E2 -19535.39} C_VEL
LIN {X 0,Y 233.255,Z 386.776,A -85,B 0,C 180,E1 -19538.667,E2 -19538.667} C_VEL
LIN {X 0,Y 233.857,Z 382.631,A -85,B 0,C 180,E1 -19541.267,E2 -19541.267} C_VEL
LIN {X 0,Y 235.045,Z 376.282,A -85,B 0,C 180,E1 -19544.284,E2 -19544.284} C_VEL
LIN {X 0,Y 236.514,Z 369.376,A -85,B 0,C 180,E1 -19546.844,E2 -19546.844} C_VEL
LIN {X 0,Y 237.992,Z 362.328,A -85,B 0,C 180,E1 -19548.958,E2 -19548.958} C_VEL
LIN {X 0,Y 239.837,Z 353.852,A -85,B 0,C 180,E1 -19551.039,E2 -19551.039} C_VEL
LIN {X 0,Y 242.092,Z 343.406,A -85,B 0,C 180,E1 -19553.076,E2 -19553.076} C_VEL
LIN {X 0,Y 242.096,Z 332.251,A -85,B 0,C 180,E1 -19554.984,E2 -19554.984} C_VEL
LIN {X 0,Y 241.791,Z 321.829,A -85,B 0,C 180,E1 -19556.461,E2 -19556.461} C_VEL
LIN {X 0,Y 240.454,Z 309.015,A -85,B 0,C 180,E1 -19558.003,E2 -19558.003} C_VEL
LIN {X 0,Y 238.427,Z 296.89,A -85,B 0,C 180,E1 -19559.206,E2 -19559.206} C_VEL
LIN {X 0,Y 235.906,Z 285.421,A -85,B 0,C 180,E1 -19560.174,E2 -19560.174} C_VEL
LIN {X 0,Y 237.388,Z 279.155,A -85,B 0,C 180,E1 -19565.264,E2 -19565.264} C_VEL
LIN {X 0,Y 237.761,Z 276.99,A -85,B 0,C 180,E1 -19567.051,E2 -19567.051} C_VEL
LIN {X 0,Y 237.617,Z 273.892,A -85,B 0,C 180,E1 -19569.736,E2 -19569.736} C_VEL
LIN {X 0,Y 236.972,Z 270.429,A -85,B 0,C 180,E1 -19573.013,E2 -19573.013} C_VEL
LIN {X 0,Y 236.032,Z 265.321,A -85,B 0,C 180,E1 -19578.11,E2 -19578.11} C_VEL
LIN {X 0,Y 235.564,Z 262.448,A -85,B 0,C 180,E1 -19581.205,E2 -19581.205} C_VEL
LIN {X 0,Y 234.945,Z 259.22,A -85,B 0,C 180,E1 -19584.968,E2 -19584.968} C_VEL
LIN {X 0,Y 234.961,Z 259.217,A -85,B 0,C 180,E1 -19587.425,E2 -19587.425} C_VEL
LIN {X 0,Y 234.91,Z 259.221,A -85,B 0,C 180,E1 -19591.401,E2 -19591.401} C_VEL
LIN {X 0,Y 234.968,Z 259.215,A -85,B 0,C 180,E1 -19595.245,E2 -19595.245} C_VEL
LIN {X 0,Y 234.977,Z 259.215,A -85,B 0,C 180,E1 -19598.967,E2 -19598.967} C_VEL
LIN {X 0,Y 235.063,Z 259.204,A -85,B 0,C 180,E1 -19603.094,E2 -19603.094} C_VEL
LIN {X 0,Y 235.093,Z 259.203,A -85,B 0,C 180,E1 -19607.921,E2 -19607.921} C_VEL
LIN {X 0,Y 235.327,Z 259.173,A -85,B 0,C 180,E1 -19611.412,E2 -19611.412} C_VEL
LIN {X 0,Y 235.375,Z 259.164,A -85,B 0,C 180,E1 -19613.141,E2 -19613.141} C_VEL
LIN {X 0,Y 235.603,Z 259.136,A -85,B 0,C 180,E1 -19618.291,E2 -19618.291} C_VEL
LIN {X 0,Y 235.589,Z 259.14,A -85,B 0,C 180,E1 -19621.71,E2 -19621.71} C_VEL
LIN {X 0,Y 235.356,Z 259.167,A -85,B 0,C 180,E1 -19626.86,E2 -19626.86} C_VEL
LIN {X 0,Y 235.221,Z 259.18,A -85,B 0,C 180,E1 -19630.327,E2 -19630.327} C_VEL
LIN {X 0,Y 235.088,Z 259.2,A -85,B 0,C 180,E1 -19635.608,E2 -19635.608} C_VEL
LIN {X 0,Y 234.995,Z 259.209,A -85,B 0,C 180,E1 -19639.207,E2 -19639.207} C_VEL
LIN {X 0,Y 234.924,Z 259.222,A -85,B 0,C 180,E1 -19642.887,E2 -19642.887} C_VEL
LIN {X 0,Y 234.931,Z 259.222,A -85,B 0,C 180,E1 -19646.662,E2 -19646.662} C_VEL
LIN {X 0,Y 234.903,Z 259.225,A -85,B 0,C 180,E1 -19650.572,E2 -19650.572} C_VEL
LIN {X 0,Y 234.938,Z 259.222,A -85,B 0,C 180,E1 -19654.637,E2 -19654.637} C_VEL
LIN {X 0,Y 234.95,Z 259.217,A -85,B 0,C 180,E1 -19658.943,E2 -19658.943} C_VEL
LIN {X 0,Y 234.885,Z 259.225,A -85,B 0,C 180,E1 -19663.487,E2 -19663.487} C_VEL
LIN {X 0,Y 234.87,Z 259.229,A -85,B 0,C 180,E1 -19666.507,E2 -19666.507} C_VEL
LIN {X 0,Y 234.925,Z 259.221,A -85,B 0,C 180,E1 -19671.077,E2 -19671.077} C_VEL
LIN {X 0,Y 234.875,Z 259.228,A -85,B 0,C 180,E1 -19675.35,E2 -19675.35} C_VEL
LIN {X 0,Y 234.843,Z 259.229,A -85,B 0,C 180,E1 -19677.404,E2 -19677.404} C_VEL
LIN {X 0,Y 234.647,Z 259.25,A -85,B 0,C 180,E1 -19679.388,E2 -19679.388} C_VEL
LIN {X 0,Y 234.586,Z 260.317,A -85,B 0,C 180,E1 -19681.355,E2 -19681.355} C_VEL
LIN {X 0,Y 234.512,Z 262.146,A -85,B 0,C 180,E1 -19684.079,E2 -19684.079} C_VEL
LIN {X 0,Y 239.322,Z 275.555,A -85,B 0,C 180,E1 -19685.556,E2 -19685.556} C_VEL
LIN {X 0,Y 242.583,Z 286.818,A -85,B 0,C 180,E1 -19686.98,E2 -19686.98} C_VEL
LIN {X 0,Y 244.921,Z 298.152,A -85,B 0,C 180,E1 -19688.597,E2 -19688.597} C_VEL
LIN {X 0,Y 245.684,Z 304.275,A -85,B 0,C 180,E1 -19689.559,E2 -19689.559} C_VEL
LIN {X 0,Y 244.016,Z 314.33,A -85,B 0,C 180,E1 -19691.092,E2 -19691.092} C_VEL
LIN {X 0,Y 241.907,Z 324.931,A -85,B 0,C 180,E1 -19693.108,E2 -19693.108} C_VEL
LIN {X 0,Y 239.892,Z 334.202,A -85,B 0,C 180,E1 -19695.327,E2 -19695.327} C_VEL
LIN {X 0,Y 238.121,Z 341.908,A -85,B 0,C 180,E1 -19697.642,E2 -19697.642} C_VEL
LIN {X 0,Y 236.665,Z 347.64,A -85,B 0,C 180,E1 -19699.734,E2 -19699.734} C_VEL
LIN {X 0,Y 235.836,Z 351.47,A -85,B 0,C 180,E1 -19701.428,E2 -19701.428} C_VEL
LIN {X 0,Y 234.77,Z 356.242,A -85,B 0,C 180,E1 -19703.983,E2 -19703.983} C_VEL
LIN {X 0,Y 233.882,Z 359.925,A -85,B 0,C 180,E1 -19706.552,E2 -19706.552} C_VEL
LIN {X 0,Y 233.532,Z 361.824,A -85,B 0,C 180,E1 -19708.273,E2 -19708.273} C_VEL
LIN {X 0,Y 233.283,Z 363.305,A -85,B 0,C 180,E1 -19709.997,E2 -19709.997} C_VEL
LIN {X 0,Y 233.198,Z 365,A -85,B 0,C 180,E1 -19713.453,E2 -19713.453} C_VEL
LIN {X 0,Y 233.341,Z 365.245,A -85,B 0,C 180,E1 -19716.313,E2 -19716.313} C_VEL
LIN {X 0,Y 233.548,Z 364.663,A -85,B 0,C 180,E1 -19718.651,E2 -19718.651} C_VEL
LIN {X 0,Y 234.319,Z 362.452,A -85,B 0,C 180,E1 -19722.117,E2 -19722.117} C_VEL
LIN {X 0,Y 235.299,Z 359.68,A -85,B 0,C 180,E1 -19724.705,E2 -19724.705} C_VEL
LIN {X 0,Y 236.63,Z 355.881,A -85,B 0,C 180,E1 -19727.275,E2 -19727.275} C_VEL
LIN {X 0,Y 238.292,Z 350.947,A -85,B 0,C 180,E1 -19729.824,E2 -19729.824} C_VEL
LIN {X 0,Y 240.415,Z 344.717,A -85,B 0,C 180,E1 -19732.332,E2 -19732.332} C_VEL
LIN {X 0,Y 242.829,Z 336.883,A -85,B 0,C 180,E1 -19734.81,E2 -19734.81} C_VEL
LIN {X 0,Y 245.09,Z 328.871,A -85,B 0,C 180,E1 -19736.846,E2 -19736.846} C_VEL
LIN {X 0,Y 247.601,Z 319.067,A -85,B 0,C 180,E1 -19738.848,E2 -19738.848} C_VEL
LIN {X 0,Y 249.567,Z 310.706,A -85,B 0,C 180,E1 -19740.221,E2 -19740.221} C_VEL
LIN {X 0,Y 248.896,Z 304.543,A -85,B 0,C 180,E1 -19741.357,E2 -19741.357} C_VEL
LIN {X 0,Y 246.755,Z 294.121,A -85,B 0,C 180,E1 -19743.157,E2 -19743.157} C_VEL
LIN {X 0,Y 243.281,Z 282.636,A -85,B 0,C 180,E1 -19744.981,E2 -19744.981} C_VEL
LIN {X 0,Y 239.413,Z 272.752,A -85,B 0,C 180,E1 -19746.465,E2 -19746.465} C_VEL
LIN {X 0,Y 236.258,Z 265.998,A -85,B 0,C 180,E1 -19747.448,E2 -19747.448} C_VEL
